KUKA KRL program: EPS_2_25716_MHDR04A_A_20260116015254.src

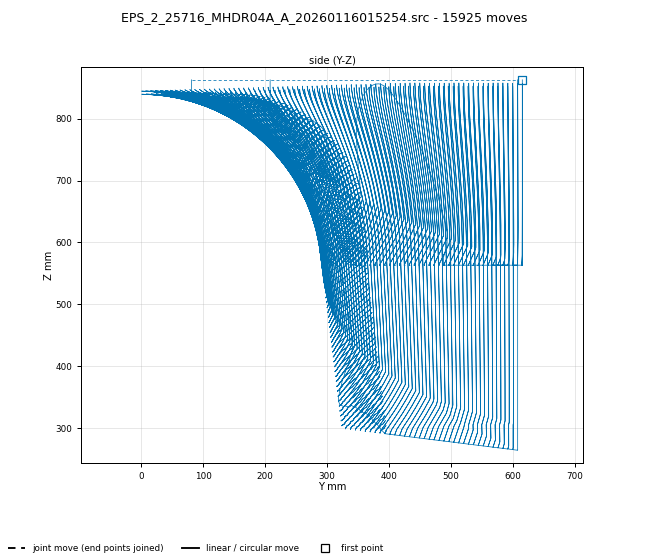
[picture p0: tool path of EPS_2_25716_MHDR04A_A_20260116015254.src, 15925 of 15927 moves have a stored position in this frame; points joined in program order, loops and branches not executed]
&ACCESS RVP
&REL 4
&COMMENT QRS 19112012
&PARAM EDITMASK = *
DEF PART()
EXT BAS (BAS_COMMAND :IN,REAL :IN )
INT I
BAS (#INITMOV,0 )

;KUKA QRS Post kuka4.cps  Date:22-06-2017 !

File_ID=2968

QRS_PRE_INIT()

;Init var - Until changes are made in qrs_pre_init
Outlet_Square_prg=0
Inlet_1_Square_prg=0
Inlet_2_Square_prg=0
Inlet_3_Square_prg=0
Inlet_4_Square_prg=0
Inlet_5_Square_prg=0

Outlet_1={X 0.000, Y 425.000, Z 586.000, B 0.000, E1 0.000 }
Inlet_1={X 0.000, Y 472.270, Z 561.000, B 0.000, E1 180.000 }
Outlet_1_type=533
Inlet_1_type=0
;QRS#1=Sidecore dimensions
;QRS#2=525-21" Concrete
;QRS#3=DeadEnd 533
;QRS#4=
;QRS#5=
;QRS#6=
;QRS#7=
;QRS#8=
;QRS#9=S306-32
;QRS#10=

;QRS#11=
;QRS#12=
;QRS#13=
;QRS#14=
;QRS#15=
;QRS#16=1220x127x1219 4'
;QRS#17=EPS Height
;QRS#18=852,5
;QRS#19=*
;QRS#20= UPDATED VERSION 22-06-2017
;QRS#21=*
Outlet_Square=0250
Inlet_1_Square=00
Inlet_2_Square=0
Inlet_3_Square=0
Inlet_4_Square=0
Inlet_5_Square=0
Mill_Square=1
Outlet_Square_Prg=263
Inlet_1_Square_prg=0

QRS_INIT()

$ADVANCE=5

; T1
PTP {E1 172.624,E2 172.624}
PTP {X 0,Y 615.399,A -85,B 0,C 180,E1 172.624,E2 172.624,E3 0,E4 0,E5 0,E6 0}
QRS_SPEED_INIT()
LIN {X 0,Y 615.399,Z 862.5,A -85,B 0,C 180,E1 172.624,E2 172.624,E3 0,E4 0,E5 0,E6 0} C_VEL
LIN {X 0,Y 615.399,Z 565.28,A -85,B 0,C 180,E1 172.624,E2 172.624} C_VEL
LIN {X 0,Y 615.426,Z 563.28,A -85,B 0,C 180,E1 172.81,E2 172.81} C_VEL
LIN {X 0,Y 615.832,Z 563.28,A -85,B 0,C 180,E1 174.193,E2 174.193} C_VEL
LIN {X 0,Y 615.876,Z 563.28,A -85,B 0,C 180,E1 178.841,E2 178.841} C_VEL
LIN {X 0,Y 615.817,Z 563.28,A -85,B 0,C 180,E1 183.48,E2 183.48} C_VEL
LIN {X 0,Y 615.805,Z 563.28,A -85,B 0,C 180,E1 188.143,E2 188.143} C_VEL
LIN {X 0,Y 615.837,Z 563.28,A -85,B 0,C 180,E1 192.861,E2 192.861} C_VEL
LIN {X 0,Y 615.756,Z 563.28,A -85,B 0,C 180,E1 197.672,E2 197.672} C_VEL
LIN {X 0,Y 615.769,Z 563.28,A -85,B 0,C 180,E1 197.99,E2 197.99} C_VEL
LIN {X 0,Y 615.763,Z 563.28,A -85,B 0,C 180,E1 202.613,E2 202.613} C_VEL
LIN {X 0,Y 615.222,Z 563.28,A -85,B 0,C 180,E1 205.173,E2 205.173} C_VEL
LIN {X 0,Y 615.704,Z 563.28,A -85,B 0,C 180,E1 207.743,E2 207.743} C_VEL
LIN {X 0,Y 615.235,Z 563.28,A -85,B 0,C 180,E1 210.422,E2 210.422} C_VEL
LIN {X 0,Y 615.861,Z 563.28,A -85,B 0,C 180,E1 213.115,E2 213.115} C_VEL
LIN {X 0,Y 615.558,Z 563.28,A -85,B 0,C 180,E1 215.95,E2 215.95} C_VEL
LIN {X 0,Y 615.606,Z 563.28,A -85,B 0,C 180,E1 217.868,E2 217.868} C_VEL
LIN {X 0,Y 615.618,Z 563.28,A -85,B 0,C 180,E1 221.912,E2 221.912} C_VEL
LIN {X 0,Y 615.192,Z 563.28,A -85,B 0,C 180,E1 225.151,E2 225.151} C_VEL
LIN {X 0,Y 615.658,Z 563.28,A -85,B 0,C 180,E1 228.093,E2 228.093} C_VEL
LIN {X 0,Y 615.552,Z 563.28,A -85,B 0,C 180,E1 232.141,E2 232.141} C_VEL
LIN {X 0,Y 615.541,Z 563.28,A -85,B 0,C 180,E1 234.05,E2 234.05} C_VEL
LIN {X 0,Y 615.711,Z 563.28,A -85,B 0,C 180,E1 236.078,E2 236.078} C_VEL
LIN {X 0,Y 615.746,Z 563.28,A -85,B 0,C 180,E1 236.879,E2 236.879} C_VEL
LIN {X 0,Y 615.823,Z 563.28,A -85,B 0,C 180,E1 240.472,E2 240.472} C_VEL
LIN {X 0,Y 615.17,Z 563.28,A -85,B 0,C 180,E1 240.877,E2 240.877} C_VEL
LIN {X 0,Y 614.627,Z 563.28,A -85,B 0,C 180,E1 240.936,E2 240.936} C_VEL
LIN {X 0,Y 614.726,Z 566.395,A -85,B 0,C 180,E1 240.996,E2 240.996} C_VEL
LIN {X 0,Y 615.379,Z 580.016,A -85,B 0,C 180,E1 241.207,E2 241.207} C_VEL
LIN {X 0,Y 615.433,Z 602.784,A -85,B 0,C 180,E1 241.52,E2 241.52} C_VEL
LIN {X 0,Y 615.521,Z 612.728,A -85,B 0,C 180,E1 241.689,E2 241.689} C_VEL
LIN {X 0,Y 615.532,Z 626.222,A -85,B 0,C 180,E1 241.976,E2 241.976} C_VEL
LIN {X 0,Y 615.495,Z 635.643,A -85,B 0,C 180,E1 242.213,E2 242.213} C_VEL
LIN {X 0,Y 615.676,Z 651.537,A -85,B 0,C 180,E1 242.706,E2 242.706} C_VEL
LIN {X 0,Y 615.645,Z 663.962,A -85,B 0,C 180,E1 243.153,E2 243.153} C_VEL
LIN {X 0,Y 615.577,Z 673.88,A -85,B 0,C 180,E1 243.555,E2 243.555} C_VEL
LIN {X 0,Y 615.711,Z 689.6,A -85,B 0,C 180,E1 244.287,E2 244.287} C_VEL
LIN {X 0,Y 615.692,Z 701.948,A -85,B 0,C 180,E1 244.936,E2 244.936} C_VEL
LIN {X 0,Y 615.677,Z 713.617,A -85,B 0,C 180,E1 245.617,E2 245.617} C_VEL
LIN {X 0,Y 615.715,Z 725.413,A -85,B 0,C 180,E1 246.38,E2 246.38} C_VEL
LIN {X 0,Y 615.721,Z 736.092,A -85,B 0,C 180,E1 247.135,E2 247.135} C_VEL
LIN {X 0,Y 615.707,Z 747.395,A -85,B 0,C 180,E1 248.012,E2 248.012} C_VEL
LIN {X 0,Y 615.704,Z 756.656,A -85,B 0,C 180,E1 248.791,E2 248.791} C_VEL
LIN {X 0,Y 615.752,Z 766.793,A -85,B 0,C 180,E1 249.723,E2 249.723} C_VEL
LIN {X 0,Y 615.723,Z 776.057,A -85,B 0,C 180,E1 250.646,E2 250.646} C_VEL
LIN {X 0,Y 615.683,Z 784.416,A -85,B 0,C 180,E1 251.548,E2 251.548} C_VEL
LIN {X 0,Y 615.766,Z 792.777,A -85,B 0,C 180,E1 252.532,E2 252.532} C_VEL
LIN {X 0,Y 615.718,Z 800.682,A -85,B 0,C 180,E1 253.542,E2 253.542} C_VEL
LIN {X 0,Y 615.581,Z 807.427,A -85,B 0,C 180,E1 254.473,E2 254.473} C_VEL
LIN {X 0,Y 615.671,Z 815.061,A -85,B 0,C 180,E1 255.645,E2 255.645} C_VEL
LIN {X 0,Y 615.807,Z 820.438,A -85,B 0,C 180,E1 256.544,E2 256.544} C_VEL
LIN {X 0,Y 615.575,Z 826.91,A -85,B 0,C 180,E1 257.728,E2 257.728} C_VEL
LIN {X 0,Y 615.616,Z 832.624,A -85,B 0,C 180,E1 258.913,E2 258.913} C_VEL
LIN {X 0,Y 615.829,Z 837.634,A -85,B 0,C 180,E1 260.096,E2 260.096} C_VEL
LIN {X 0,Y 615.604,Z 842.064,A -85,B 0,C 180,E1 261.268,E2 261.268} C_VEL
LIN {X 0,Y 615.654,Z 846.465,A -85,B 0,C 180,E1 262.658,E2 262.658} C_VEL
LIN {X 0,Y 615.788,Z 849.368,A -85,B 0,C 180,E1 263.749,E2 263.749} C_VEL
LIN {X 0,Y 615.542,Z 852.381,A -85,B 0,C 180,E1 265.123,E2 265.123} C_VEL
LIN {X 0,Y 615.642,Z 854.591,A -85,B 0,C 180,E1 266.519,E2 266.519} C_VEL
LIN {X 0,Y 615.833,Z 855.667,A -85,B 0,C 180,E1 267.449,E2 267.449} C_VEL
LIN {X 0,Y 615.553,Z 856.715,A -85,B 0,C 180,E1 268.84,E2 268.84} C_VEL
LIN {X 0,Y 615.842,Z 856.659,A -85,B 0,C 180,E1 271.159,E2 271.159} C_VEL
LIN {X 0,Y 615.567,Z 855.717,A -85,B 0,C 180,E1 272.552,E2 272.552} C_VEL
LIN {X 0,Y 615.55,Z 854.608,A -85,B 0,C 180,E1 273.482,E2 273.482} C_VEL
LIN {X 0,Y 615.828,Z 852.329,A -85,B 0,C 180,E1 274.875,E2 274.875} C_VEL
LIN {X 0,Y 615.615,Z 849.405,A -85,B 0,C 180,E1 276.251,E2 276.251} C_VEL
LIN {X 0,Y 615.622,Z 846.265,A -85,B 0,C 180,E1 277.419,E2 277.419} C_VEL
LIN {X 0,Y 615.784,Z 842.036,A -85,B 0,C 180,E1 278.729,E2 278.729} C_VEL
LIN {X 0,Y 615.572,Z 837.671,A -85,B 0,C 180,E1 279.908,E2 279.908} C_VEL
LIN {X 0,Y 615.632,Z 832.622,A -85,B 0,C 180,E1 281.086,E2 281.086} C_VEL
LIN {X 0,Y 615.805,Z 826.883,A -85,B 0,C 180,E1 282.267,E2 282.267} C_VEL
LIN {X 0,Y 615.626,Z 820.456,A -85,B 0,C 180,E1 283.46,E2 283.46} C_VEL
LIN {X 0,Y 615.698,Z 813.195,A -85,B 0,C 180,E1 284.654,E2 284.654} C_VEL
LIN {X 0,Y 615.811,Z 807.631,A -85,B 0,C 180,E1 285.488,E2 285.488} C_VEL
LIN {X 0,Y 615.663,Z 798.199,A -85,B 0,C 180,E1 286.791,E2 286.791} C_VEL
LIN {X 0,Y 615.737,Z 789.606,A -85,B 0,C 180,E1 287.852,E2 287.852} C_VEL
LIN {X 0,Y 615.77,Z 781.414,A -85,B 0,C 180,E1 288.784,E2 288.784} C_VEL
LIN {X 0,Y 615.697,Z 771.526,A -85,B 0,C 180,E1 289.816,E2 289.816} C_VEL
LIN {X 0,Y 615.715,Z 763.539,A -85,B 0,C 180,E1 290.588,E2 290.588} C_VEL
LIN {X 0,Y 615.746,Z 753.036,A -85,B 0,C 180,E1 291.518,E2 291.518} C_VEL
LIN {X 0,Y 615.704,Z 743.049,A -85,B 0,C 180,E1 292.335,E2 292.335} C_VEL
LIN {X 0,Y 615.702,Z 733.298,A -85,B 0,C 180,E1 293.071,E2 293.071} C_VEL
LIN {X 0,Y 615.683,Z 721.635,A -85,B 0,C 180,E1 293.874,E2 293.874} C_VEL
LIN {X 0,Y 615.698,Z 709.596,A -85,B 0,C 180,E1 294.623,E2 294.623} C_VEL
LIN {X 0,Y 615.649,Z 698.891,A -85,B 0,C 180,E1 295.234,E2 295.234} C_VEL
LIN {X 0,Y 615.644,Z 688.027,A -85,B 0,C 180,E1 295.796,E2 295.796} C_VEL
LIN {X 0,Y 615.702,Z 673.88,A -85,B 0,C 180,E1 296.439,E2 296.439} C_VEL
LIN {X 0,Y 615.617,Z 660.684,A -85,B 0,C 180,E1 296.971,E2 296.971} C_VEL
LIN {X 0,Y 615.56,Z 651.537,A -85,B 0,C 180,E1 297.299,E2 297.299} C_VEL
LIN {X 0,Y 615.62,Z 634.846,A -85,B 0,C 180,E1 297.801,E2 297.801} C_VEL
LIN {X 0,Y 615.416,Z 621.524,A -85,B 0,C 180,E1 298.137,E2 298.137} C_VEL
LIN {X 0,Y 615.596,Z 607.658,A -85,B 0,C 180,E1 298.397,E2 298.397} C_VEL
LIN {X 0,Y 615.505,Z 590.993,A -85,B 0,C 180,E1 298.643,E2 298.643} C_VEL
LIN {X 0,Y 615.29,Z 577.557,A -85,B 0,C 180,E1 298.829,E2 298.829} C_VEL
LIN {X 0,Y 614.571,Z 564.121,A -85,B 0,C 180,E1 299.042,E2 299.042} C_VEL
LIN {X 0,Y 614.836,Z 563.28,A -85,B 0,C 180,E1 299.087,E2 299.087} C_VEL
LIN {X 0,Y 615.174,Z 563.28,A -85,B 0,C 180,E1 299.128,E2 299.128} C_VEL
LIN {X 0,Y 615.852,Z 563.28,A -85,B 0,C 180,E1 299.532,E2 299.532} C_VEL
LIN {X 0,Y 615.848,Z 563.28,A -85,B 0,C 180,E1 300.387,E2 300.387} C_VEL
LIN {X 0,Y 615.152,Z 563.28,A -85,B 0,C 180,E1 303.844,E2 303.844} C_VEL
LIN {X 0,Y 615.705,Z 563.28,A -85,B 0,C 180,E1 305.939,E2 305.939} C_VEL
LIN {X 0,Y 615.725,Z 563.28,A -85,B 0,C 180,E1 308.857,E2 308.857} C_VEL
LIN {X 0,Y 615.233,Z 563.28,A -85,B 0,C 180,E1 311.942,E2 311.942} C_VEL
LIN {X 0,Y 615.67,Z 563.28,A -85,B 0,C 180,E1 314.894,E2 314.894} C_VEL
LIN {X 0,Y 615.636,Z 563.28,A -85,B 0,C 180,E1 318.496,E2 318.496} C_VEL
LIN {X 0,Y 615.343,Z 563.28,A -85,B 0,C 180,E1 321.113,E2 321.113} C_VEL
LIN {X 0,Y 615.391,Z 563.28,A -85,B 0,C 180,E1 322.158,E2 322.158} C_VEL
LIN {X 0,Y 615.635,Z 563.28,A -85,B 0,C 180,E1 324.055,E2 324.055} C_VEL
LIN {X 0,Y 615.105,Z 563.28,A -85,B 0,C 180,E1 326.839,E2 326.839} C_VEL
LIN {X 0,Y 615.706,Z 563.28,A -85,B 0,C 180,E1 329.604,E2 329.604} C_VEL
LIN {X 0,Y 615.206,Z 563.28,A -85,B 0,C 180,E1 332.233,E2 332.233} C_VEL
LIN {X 0,Y 615.75,Z 563.28,A -85,B 0,C 180,E1 334.85,E2 334.85} C_VEL
LIN {X 0,Y 615.758,Z 563.28,A -85,B 0,C 180,E1 339.877,E2 339.877} C_VEL
LIN {X 0,Y 615.78,Z 563.28,A -85,B 0,C 180,E1 343.784,E2 343.784} C_VEL
LIN {X 0,Y 615.808,Z 563.28,A -85,B 0,C 180,E1 349.507,E2 349.507} C_VEL
LIN {X 0,Y 615.82,Z 563.28,A -85,B 0,C 180,E1 354.193,E2 354.193} C_VEL
LIN {X 0,Y 615.861,Z 563.28,A -85,B 0,C 180,E1 358.841,E2 358.841} C_VEL
LIN {X 0,Y 615.87,Z 563.28,A -85,B 0,C 180,E1 363.48,E2 363.48} C_VEL
LIN {X 0,Y 615.8,Z 563.28,A -85,B 0,C 180,E1 368.143,E2 368.143} C_VEL
LIN {X 0,Y 615.811,Z 563.28,A -85,B 0,C 180,E1 372.861,E2 372.861} C_VEL
LIN {X 0,Y 615.81,Z 563.28,A -85,B 0,C 180,E1 377.67,E2 377.67} C_VEL
LIN {X 0,Y 615.807,Z 563.28,A -85,B 0,C 180,E1 378.001,E2 378.001} C_VEL
LIN {X 0,Y 615.761,Z 563.28,A -85,B 0,C 180,E1 382.613,E2 382.613} C_VEL
LIN {X 0,Y 615.227,Z 563.28,A -85,B 0,C 180,E1 385.173,E2 385.173} C_VEL
LIN {X 0,Y 615.728,Z 563.28,A -85,B 0,C 180,E1 387.742,E2 387.742} C_VEL
LIN {X 0,Y 615.24,Z 563.28,A -85,B 0,C 180,E1 390.422,E2 390.422} C_VEL
LIN {X 0,Y 615.85,Z 563.28,A -85,B 0,C 180,E1 393.116,E2 393.116} C_VEL
LIN {X 0,Y 615.533,Z 563.28,A -85,B 0,C 180,E1 395.952,E2 395.952} C_VEL
LIN {X 0,Y 615.606,Z 563.28,A -85,B 0,C 180,E1 397.868,E2 397.868} C_VEL
LIN {X 0,Y 615.685,Z 563.28,A -85,B 0,C 180,E1 401.906,E2 401.906} C_VEL
LIN {X 0,Y 615.223,Z 563.28,A -85,B 0,C 180,E1 405.148,E2 405.148} C_VEL
LIN {X 0,Y 615.683,Z 563.28,A -85,B 0,C 180,E1 408.095,E2 408.095} C_VEL
LIN {X 0,Y 615.591,Z 563.28,A -85,B 0,C 180,E1 412.136,E2 412.136} C_VEL
LIN {X 0,Y 615.556,Z 563.28,A -85,B 0,C 180,E1 414.051,E2 414.051} C_VEL
LIN {X 0,Y 615.726,Z 563.28,A -85,B 0,C 180,E1 416.076,E2 416.076} C_VEL
LIN {X 0,Y 615.719,Z 563.28,A -85,B 0,C 180,E1 416.878,E2 416.878} C_VEL
LIN {X 0,Y 615.543,Z 563.28,A -85,B 0,C 180,E1 420.519,E2 420.519} C_VEL
LIN {X 0,Y 615.508,Z 563.28,A -85,B 0,C 180,E1 422.249,E2 422.249} C_VEL
LIN {X 0,Y 615.423,Z 563.28,A -85,B 0,C 180,E1 425.669,E2 425.669} C_VEL
LIN {X 0,Y 615.587,Z 563.28,A -85,B 0,C 180,E1 427.381,E2 427.381} C_VEL
LIN {X 0,Y 615.807,Z 563.28,A -85,B 0,C 180,E1 432.005,E2 432.005} C_VEL
LIN {X 0,Y 615.812,Z 563.28,A -85,B 0,C 180,E1 432.331,E2 432.331} C_VEL
LIN {X 0,Y 615.818,Z 563.28,A -85,B 0,C 180,E1 437.139,E2 437.139} C_VEL
LIN {X 0,Y 615.845,Z 563.28,A -85,B 0,C 180,E1 441.857,E2 441.857} C_VEL
LIN {X 0,Y 615.853,Z 563.28,A -85,B 0,C 180,E1 446.52,E2 446.52} C_VEL
LIN {X 0,Y 615.874,Z 563.28,A -85,B 0,C 180,E1 451.159,E2 451.159} C_VEL
LIN {X 0,Y 615.861,Z 563.28,A -85,B 0,C 180,E1 455.806,E2 455.806} C_VEL
LIN {X 0,Y 615.821,Z 563.28,A -85,B 0,C 180,E1 460.493,E2 460.493} C_VEL
LIN {X 0,Y 615.809,Z 563.28,A -85,B 0,C 180,E1 465.251,E2 465.251} C_VEL
LIN {X 0,Y 615.79,Z 563.28,A -85,B 0,C 180,E1 470.121,E2 470.121} C_VEL
LIN {X 0,Y 615.764,Z 563.28,A -85,B 0,C 180,E1 475.149,E2 475.149} C_VEL
LIN {X 0,Y 615.395,Z 563.28,A -85,B 0,C 180,E1 479.457,E2 479.457} C_VEL
LIN {X 0,Y 615.72,Z 563.28,A -85,B 0,C 180,E1 480.394,E2 480.394} C_VEL
LIN {X 0,Y 615.148,Z 563.28,A -85,B 0,C 180,E1 483.844,E2 483.844} C_VEL
LIN {X 0,Y 615.695,Z 563.28,A -85,B 0,C 180,E1 485.939,E2 485.939} C_VEL
LIN {X 0,Y 615.655,Z 563.28,A -85,B 0,C 180,E1 487.871,E2 487.871} C_VEL
LIN {X 0,Y 615.739,Z 563.28,A -85,B 0,C 180,E1 488.856,E2 488.856} C_VEL
LIN {X 0,Y 615.245,Z 563.28,A -85,B 0,C 180,E1 491.941,E2 491.941} C_VEL
LIN {X 0,Y 615.675,Z 563.28,A -85,B 0,C 180,E1 494.895,E2 494.895} C_VEL
LIN {X 0,Y 615.643,Z 563.28,A -85,B 0,C 180,E1 498.495,E2 498.495} C_VEL
LIN {X 0,Y 615.366,Z 563.28,A -85,B 0,C 180,E1 501.115,E2 501.115} C_VEL
LIN {X 0,Y 615.411,Z 563.28,A -85,B 0,C 180,E1 502.155,E2 502.155} C_VEL
LIN {X 0,Y 615.682,Z 563.28,A -85,B 0,C 180,E1 504.059,E2 504.059} C_VEL
LIN {X 0,Y 615.129,Z 563.28,A -85,B 0,C 180,E1 506.841,E2 506.841} C_VEL
LIN {X 0,Y 615.712,Z 563.28,A -85,B 0,C 180,E1 509.604,E2 509.604} C_VEL
LIN {X 0,Y 615.229,Z 563.28,A -85,B 0,C 180,E1 512.234,E2 512.234} C_VEL
LIN {X 0,Y 615.78,Z 563.28,A -85,B 0,C 180,E1 514.851,E2 514.851} C_VEL
LIN {X 0,Y 615.783,Z 563.28,A -85,B 0,C 180,E1 519.878,E2 519.878} C_VEL
LIN {X 0,Y 615.72,Z 563.28,A -85,B 0,C 180,E1 523.298,E2 523.298} C_VEL
LIN {X 0,Y 615.386,Z 563.28,A -85,B 0,C 180,E1 524.737,E2 524.737} C_VEL
LIN {X 0,Y 615.804,Z 563.28,A -85,B 0,C 180,E1 529.507,E2 529.507} C_VEL
LIN {X 0,Y 615.426,Z 563.28,A -85,B 0,C 180,E1 532.81,E2 532.81} C_VEL
LIN {X 0,Y 613.004,Z 563.28,A -85,B 0,C 180,E1 534.012,E2 534.012} C_VEL
LIN {X 0,Y 607.591,Z 563.28,A -85,B 0,C 180,E1 535.809,E2 535.809} C_VEL
LIN {X 0,Y 607.482,Z 563.28,A -85,B 0,C 180,E1 536.017,E2 536.017} C_VEL
LIN {X 0,Y 607.61,Z 563.28,A -85,B 0,C 180,E1 539.999,E2 539.999} C_VEL
LIN {X 0,Y 607.656,Z 563.28,A -85,B 0,C 180,E1 544.271,E2 544.271} C_VEL
LIN {X 0,Y 607.76,Z 563.28,A -85,B 0,C 180,E1 548.566,E2 548.566} C_VEL
LIN {X 0,Y 607.927,Z 563.28,A -85,B 0,C 180,E1 552.907,E2 552.907} C_VEL
LIN {X 0,Y 607.596,Z 563.28,A -85,B 0,C 180,E1 558.834,E2 558.834} C_VEL
LIN {X 0,Y 607.579,Z 563.28,A -85,B 0,C 180,E1 563.413,E2 563.413} C_VEL
LIN {X 0,Y 607.666,Z 563.28,A -85,B 0,C 180,E1 568.151,E2 568.151} C_VEL
LIN {X 0,Y 607.954,Z 563.28,A -85,B 0,C 180,E1 573.095,E2 573.095} C_VEL
LIN {X 0,Y 607.552,Z 563.28,A -85,B 0,C 180,E1 578.382,E2 578.382} C_VEL
LIN {X 0,Y 607.644,Z 563.28,A -85,B 0,C 180,E1 582.104,E2 582.104} C_VEL
LIN {X 0,Y 607.732,Z 563.28,A -85,B 0,C 180,E1 588.148,E2 588.148} C_VEL
LIN {X 0,Y 607.577,Z 563.28,A -85,B 0,C 180,E1 593.41,E2 593.41} C_VEL
LIN {X 0,Y 607.682,Z 563.28,A -85,B 0,C 180,E1 597.592,E2 597.592} C_VEL
LIN {X 0,Y 607.69,Z 563.28,A -85,B 0,C 180,E1 600.567,E2 600.567} C_VEL
LIN {X 0,Y 608.559,Z 624.797,A -85,B 0,C 180,E1 601.589,E2 601.589} C_VEL
LIN {X 0,Y 608.498,Z 665.533,A -85,B 0,C 180,E1 602.876,E2 602.876} C_VEL
LIN {X 0,Y 608.385,Z 702.866,A -85,B 0,C 180,E1 604.667,E2 604.667} C_VEL
LIN {X 0,Y 608.235,Z 738.17,A -85,B 0,C 180,E1 606.998,E2 606.998} C_VEL
LIN {X 0,Y 608.103,Z 768.949,A -85,B 0,C 180,E1 609.67,E2 609.67} C_VEL
LIN {X 0,Y 608.003,Z 795.695,A -85,B 0,C 180,E1 612.672,E2 612.672} C_VEL
LIN {X 0,Y 607.895,Z 818.344,A -85,B 0,C 180,E1 615.993,E2 615.993} C_VEL
LIN {X 0,Y 607.88,Z 836.513,A -85,B 0,C 180,E1 619.631,E2 619.631} C_VEL
LIN {X 0,Y 607.848,Z 848.574,A -85,B 0,C 180,E1 623.205,E2 623.205} C_VEL
LIN {X 0,Y 607.671,Z 853.956,A -85,B 0,C 180,E1 625.727,E2 625.727} C_VEL
LIN {X 0,Y 607.708,Z 857.086,A -85,B 0,C 180,E1 628.576,E2 628.576} C_VEL
LIN {X 0,Y 607.886,Z 857.087,A -85,B 0,C 180,E1 631.422,E2 631.422} C_VEL
LIN {X 0,Y 607.927,Z 852.758,A -85,B 0,C 180,E1 634.983,E2 634.983} C_VEL
LIN {X 0,Y 607.878,Z 842.075,A -85,B 0,C 180,E1 638.925,E2 638.925} C_VEL
LIN {X 0,Y 607.906,Z 826.455,A -85,B 0,C 180,E1 642.544,E2 642.544} C_VEL
LIN {X 0,Y 607.957,Z 805.351,A -85,B 0,C 180,E1 646.029,E2 646.029} C_VEL
LIN {X 0,Y 608.034,Z 779.03,A -85,B 0,C 180,E1 649.289,E2 649.289} C_VEL
LIN {X 0,Y 608.171,Z 749.03,A -85,B 0,C 180,E1 652.137,E2 652.137} C_VEL
LIN {X 0,Y 608.315,Z 715.907,A -85,B 0,C 180,E1 654.551,E2 654.551} C_VEL
LIN {X 0,Y 608.48,Z 679.749,A -85,B 0,C 180,E1 656.512,E2 656.512} C_VEL
LIN {X 0,Y 608.582,Z 643.016,A -85,B 0,C 180,E1 657.91,E2 657.91} C_VEL
LIN {X 0,Y 608.637,Z 607.158,A -85,B 0,C 180,E1 658.759,E2 658.759} C_VEL
LIN {X 0,Y 607.764,Z 563.28,A -85,B 0,C 180,E1 659.466,E2 659.466} C_VEL
LIN {X 0,Y 607.703,Z 563.28,A -85,B 0,C 180,E1 666.58,E2 666.58} C_VEL
LIN {X 0,Y 607.312,Z 563.28,A -85,B 0,C 180,E1 672.134,E2 672.134} C_VEL
LIN {X 0,Y 607.571,Z 563.28,A -85,B 0,C 180,E1 677.89,E2 677.89} C_VEL
LIN {X 0,Y 607.598,Z 563.28,A -85,B 0,C 180,E1 683.415,E2 683.415} C_VEL
LIN {X 0,Y 607.539,Z 563.28,A -85,B 0,C 180,E1 690.38,E2 690.38} C_VEL
LIN {X 0,Y 607.785,Z 563.28,A -85,B 0,C 180,E1 695.036,E2 695.036} C_VEL
LIN {X 0,Y 607.555,Z 563.28,A -85,B 0,C 180,E1 701.164,E2 701.164} C_VEL
LIN {X 0,Y 607.221,Z 563.28,A -85,B 0,C 180,E1 705.612,E2 705.612} C_VEL
LIN {X 0,Y 607.733,Z 563.28,A -85,B 0,C 180,E1 709.992,E2 709.992} C_VEL
LIN {X 0,Y 607.882,Z 563.28,A -85,B 0,C 180,E1 714.303,E2 714.303} C_VEL
LIN {X 0,Y 607.584,Z 563.28,A -85,B 0,C 180,E1 720.001,E2 720.001} C_VEL
LIN {X 0,Y 607.669,Z 563.28,A -85,B 0,C 180,E1 724.274,E2 724.274} C_VEL
LIN {X 0,Y 607.757,Z 563.28,A -85,B 0,C 180,E1 728.569,E2 728.569} C_VEL
LIN {X 0,Y 607.883,Z 563.28,A -85,B 0,C 180,E1 732.911,E2 732.911} C_VEL
LIN {X 0,Y 607.601,Z 563.28,A -85,B 0,C 180,E1 738.837,E2 738.837} C_VEL
LIN {X 0,Y 607.579,Z 563.28,A -85,B 0,C 180,E1 743.416,E2 743.416} C_VEL
LIN {X 0,Y 607.674,Z 563.28,A -85,B 0,C 180,E1 748.154,E2 748.154} C_VEL
LIN {X 0,Y 607.942,Z 563.28,A -85,B 0,C 180,E1 753.099,E2 753.099} C_VEL
LIN {X 0,Y 607.564,Z 563.28,A -85,B 0,C 180,E1 758.385,E2 758.385} C_VEL
LIN {X 0,Y 607.717,Z 563.28,A -85,B 0,C 180,E1 762.102,E2 762.102} C_VEL
LIN {X 0,Y 607.766,Z 563.28,A -85,B 0,C 180,E1 768.149,E2 768.149} C_VEL
LIN {X 0,Y 607.616,Z 563.28,A -85,B 0,C 180,E1 773.414,E2 773.414} C_VEL
LIN {X 0,Y 607.597,Z 563.28,A -85,B 0,C 180,E1 777.61,E2 777.61} C_VEL
LIN {X 0,Y 607.587,Z 563.28,A -85,B 0,C 180,E1 781.844,E2 781.844} C_VEL
LIN {X 0,Y 607.461,Z 563.28,A -85,B 0,C 180,E1 788.123,E2 788.123} C_VEL
LIN {X 0,Y 607.79,Z 563.28,A -85,B 0,C 180,E1 792.667,E2 792.667} C_VEL
LIN {X 0,Y 607.89,Z 563.28,A -85,B 0,C 180,E1 797.091,E2 797.091} C_VEL
LIN {X 0,Y 607.6,Z 563.28,A -85,B 0,C 180,E1 802.867,E2 802.867} C_VEL
LIN {X 0,Y 607.729,Z 563.28,A -85,B 0,C 180,E1 807.154,E2 807.154} C_VEL
LIN {X 0,Y 607.865,Z 563.28,A -85,B 0,C 180,E1 811.423,E2 811.423} C_VEL
LIN {X 0,Y 607.66,Z 563.28,A -85,B 0,C 180,E1 816.619,E2 816.619} C_VEL
LIN {X 0,Y 607.592,Z 563.28,A -85,B 0,C 180,E1 821.461,E2 821.461} C_VEL
LIN {X 0,Y 607.662,Z 563.28,A -85,B 0,C 180,E1 825.853,E2 825.853} C_VEL
LIN {X 0,Y 607.792,Z 563.28,A -85,B 0,C 180,E1 830.341,E2 830.341} C_VEL
LIN {X 0,Y 607.801,Z 563.28,A -85,B 0,C 180,E1 834.966,E2 834.966} C_VEL
LIN {X 0,Y 607.608,Z 563.28,A -85,B 0,C 180,E1 839.783,E2 839.783} C_VEL
LIN {X 0,Y 607.725,Z 563.28,A -85,B 0,C 180,E1 846.58,E2 846.58} C_VEL
LIN {X 0,Y 607.33,Z 563.28,A -85,B 0,C 180,E1 851.805,E2 851.805} C_VEL
LIN {X 0,Y 607.496,Z 563.28,A -85,B 0,C 180,E1 856.085,E2 856.085} C_VEL
LIN {X 0,Y 607.415,Z 563.28,A -85,B 0,C 180,E1 860.367,E2 860.367} C_VEL
LIN {X 0,Y 607.409,Z 563.28,A -85,B 0,C 180,E1 865.151,E2 865.151} C_VEL
LIN {X 0,Y 607.556,Z 563.28,A -85,B 0,C 180,E1 870.38,E2 870.38} C_VEL
LIN {X 0,Y 607.802,Z 563.28,A -85,B 0,C 180,E1 875.034,E2 875.034} C_VEL
LIN {X 0,Y 607.616,Z 563.28,A -85,B 0,C 180,E1 881.163,E2 881.163} C_VEL
LIN {X 0,Y 607.226,Z 563.28,A -85,B 0,C 180,E1 885.742,E2 885.742} C_VEL
LIN {X 0,Y 607.733,Z 563.28,A -85,B 0,C 180,E1 889.989,E2 889.989} C_VEL
LIN {X 0,Y 607.888,Z 563.28,A -85,B 0,C 180,E1 894.3,E2 894.3} C_VEL
LIN {X 0,Y 607.482,Z 563.28,A -85,B 0,C 180,E1 896.017,E2 896.017} C_VEL
LIN {X 0,Y 603.689,Z 563.28,A -85,B 0,C 180,E1 897.629,E2 897.629} C_VEL
LIN {X 0,Y 599.797,Z 563.28,A -85,B 0,C 180,E1 899.261,E2 899.261} C_VEL
LIN {X 0,Y 599.738,Z 563.28,A -85,B 0,C 180,E1 904.327,E2 904.327} C_VEL
LIN {X 0,Y 599.818,Z 563.28,A -85,B 0,C 180,E1 908.68,E2 908.68} C_VEL
LIN {X 0,Y 599.947,Z 563.28,A -85,B 0,C 180,E1 913.082,E2 913.082} C_VEL
LIN {X 0,Y 599.642,Z 563.28,A -85,B 0,C 180,E1 919.094,E2 919.094} C_VEL
LIN {X 0,Y 599.586,Z 563.28,A -85,B 0,C 180,E1 923.744,E2 923.744} C_VEL
LIN {X 0,Y 599.666,Z 563.28,A -85,B 0,C 180,E1 928.56,E2 928.56} C_VEL
LIN {X 0,Y 599.835,Z 563.28,A -85,B 0,C 180,E1 933.881,E2 933.881} C_VEL
LIN {X 0,Y 599.527,Z 563.28,A -85,B 0,C 180,E1 938.992,E2 938.992} C_VEL
LIN {X 0,Y 599.438,Z 563.28,A -85,B 0,C 180,E1 943.109,E2 943.109} C_VEL
LIN {X 0,Y 599.557,Z 563.28,A -85,B 0,C 180,E1 949.126,E2 949.126} C_VEL
LIN {X 0,Y 599.682,Z 563.28,A -85,B 0,C 180,E1 954.636,E2 954.636} C_VEL
LIN {X 0,Y 599.928,Z 563.28,A -85,B 0,C 180,E1 960.161,E2 960.161} C_VEL
LIN {X 0,Y 601.599,Z 583.884,A -85,B 0,C 180,E1 960.536,E2 960.536} C_VEL
LIN {X 0,Y 601.567,Z 627.343,A -85,B 0,C 180,E1 961.294,E2 961.294} C_VEL
LIN {X 0,Y 601.381,Z 666.029,A -85,B 0,C 180,E1 962.549,E2 962.549} C_VEL
LIN {X 0,Y 601.087,Z 702.885,A -85,B 0,C 180,E1 964.338,E2 964.338} C_VEL
LIN {X 0,Y 600.762,Z 737.804,A -85,B 0,C 180,E1 966.666,E2 966.666} C_VEL
LIN {X 0,Y 600.476,Z 768.952,A -85,B 0,C 180,E1 969.4,E2 969.4} C_VEL
LIN {X 0,Y 600.274,Z 795.697,A -85,B 0,C 180,E1 972.442,E2 972.442} C_VEL
LIN {X 0,Y 600.064,Z 818.354,A -85,B 0,C 180,E1 975.808,E2 975.808} C_VEL
LIN {X 0,Y 599.962,Z 835.869,A -85,B 0,C 180,E1 979.338,E2 979.338} C_VEL
LIN {X 0,Y 599.89,Z 847.677,A -85,B 0,C 180,E1 982.774,E2 982.774} C_VEL
LIN {X 0,Y 599.784,Z 853.958,A -85,B 0,C 180,E1 985.671,E2 985.671} C_VEL
LIN {X 0,Y 599.809,Z 857.088,A -85,B 0,C 180,E1 988.558,E2 988.558} C_VEL
LIN {X 0,Y 599.979,Z 857.088,A -85,B 0,C 180,E1 991.441,E2 991.441} C_VEL
LIN {X 0,Y 600.013,Z 852.757,A -85,B 0,C 180,E1 995.049,E2 995.049} C_VEL
LIN {X 0,Y 599.977,Z 842.076,A -85,B 0,C 180,E1 999.043,E2 999.043} C_VEL
LIN {X 0,Y 600.04,Z 826.459,A -85,B 0,C 180,E1 1002.711,E2 1002.711} C_VEL
LIN {X 0,Y 600.116,Z 804.713,A -85,B 0,C 180,E1 1006.334,E2 1006.334} C_VEL
LIN {X 0,Y 600.366,Z 779.034,A -85,B 0,C 180,E1 1009.545,E2 1009.545} C_VEL
LIN {X 0,Y 600.648,Z 748.454,A -85,B 0,C 180,E1 1012.479,E2 1012.479} C_VEL
LIN {X 0,Y 601.003,Z 713.913,A -85,B 0,C 180,E1 1015,E2 1015} C_VEL
LIN {X 0,Y 601.367,Z 675.827,A -85,B 0,C 180,E1 1017.037,E2 1017.037} C_VEL
LIN {X 0,Y 601.573,Z 636.508,A -85,B 0,C 180,E1 1018.463,E2 1018.463} C_VEL
LIN {X 0,Y 601.717,Z 596.802,A -85,B 0,C 180,E1 1019.285,E2 1019.285} C_VEL
LIN {X 0,Y 600.038,Z 563.28,A -85,B 0,C 180,E1 1019.835,E2 1019.835} C_VEL
LIN {X 0,Y 599.744,Z 563.28,A -85,B 0,C 180,E1 1027.146,E2 1027.146} C_VEL
LIN {X 0,Y 599.412,Z 563.28,A -85,B 0,C 180,E1 1033.111,E2 1033.111} C_VEL
LIN {X 0,Y 599.576,Z 563.28,A -85,B 0,C 180,E1 1039.028,E2 1039.028} C_VEL
LIN {X 0,Y 599.521,Z 563.28,A -85,B 0,C 180,E1 1044.628,E2 1044.628} C_VEL
LIN {X 0,Y 599.594,Z 563.28,A -85,B 0,C 180,E1 1049.781,E2 1049.781} C_VEL
LIN {X 0,Y 599.852,Z 563.28,A -85,B 0,C 180,E1 1054.907,E2 1054.907} C_VEL
LIN {X 0,Y 599.708,Z 563.28,A -85,B 0,C 180,E1 1060.908,E2 1060.908} C_VEL
LIN {X 0,Y 599.36,Z 563.28,A -85,B 0,C 180,E1 1065.42,E2 1065.42} C_VEL
LIN {X 0,Y 599.793,Z 563.28,A -85,B 0,C 180,E1 1069.858,E2 1069.858} C_VEL
LIN {X 0,Y 599.981,Z 563.28,A -85,B 0,C 180,E1 1074.228,E2 1074.228} C_VEL
LIN {X 0,Y 599.684,Z 563.28,A -85,B 0,C 180,E1 1080.002,E2 1080.002} C_VEL
LIN {X 0,Y 599.751,Z 563.28,A -85,B 0,C 180,E1 1084.33,E2 1084.33} C_VEL
LIN {X 0,Y 599.811,Z 563.28,A -85,B 0,C 180,E1 1088.683,E2 1088.683} C_VEL
LIN {X 0,Y 599.909,Z 563.28,A -85,B 0,C 180,E1 1093.086,E2 1093.086} C_VEL
LIN {X 0,Y 599.661,Z 563.28,A -85,B 0,C 180,E1 1099.096,E2 1099.096} C_VEL
LIN {X 0,Y 599.587,Z 563.28,A -85,B 0,C 180,E1 1103.747,E2 1103.747} C_VEL
LIN {X 0,Y 599.675,Z 563.28,A -85,B 0,C 180,E1 1108.563,E2 1108.563} C_VEL
LIN {X 0,Y 599.823,Z 563.28,A -85,B 0,C 180,E1 1113.882,E2 1113.882} C_VEL
LIN {X 0,Y 599.534,Z 563.28,A -85,B 0,C 180,E1 1118.995,E2 1118.995} C_VEL
LIN {X 0,Y 599.493,Z 563.28,A -85,B 0,C 180,E1 1123.117,E2 1123.117} C_VEL
LIN {X 0,Y 599.571,Z 563.28,A -85,B 0,C 180,E1 1129.129,E2 1129.129} C_VEL
LIN {X 0,Y 599.715,Z 563.28,A -85,B 0,C 180,E1 1134.64,E2 1134.64} C_VEL
LIN {X 0,Y 599.597,Z 563.28,A -85,B 0,C 180,E1 1139.779,E2 1139.779} C_VEL
LIN {X 0,Y 599.484,Z 563.28,A -85,B 0,C 180,E1 1144.985,E2 1144.985} C_VEL
LIN {X 0,Y 599.394,Z 563.28,A -85,B 0,C 180,E1 1149.363,E2 1149.363} C_VEL
LIN {X 0,Y 599.552,Z 563.28,A -85,B 0,C 180,E1 1153.928,E2 1153.928} C_VEL
LIN {X 0,Y 599.636,Z 563.28,A -85,B 0,C 180,E1 1158.386,E2 1158.386} C_VEL
LIN {X 0,Y 599.702,Z 563.28,A -85,B 0,C 180,E1 1162.773,E2 1162.773} C_VEL
LIN {X 0,Y 599.84,Z 563.28,A -85,B 0,C 180,E1 1167.117,E2 1167.117} C_VEL
LIN {X 0,Y 599.955,Z 563.28,A -85,B 0,C 180,E1 1171.442,E2 1171.442} C_VEL
LIN {X 0,Y 600.029,Z 563.28,A -85,B 0,C 180,E1 1175.774,E2 1175.774} C_VEL
LIN {X 0,Y 599.651,Z 563.28,A -85,B 0,C 180,E1 1181.615,E2 1181.615} C_VEL
LIN {X 0,Y 599.504,Z 563.28,A -85,B 0,C 180,E1 1186.96,E2 1186.96} C_VEL
LIN {X 0,Y 599.564,Z 563.28,A -85,B 0,C 180,E1 1191.371,E2 1191.371} C_VEL
LIN {X 0,Y 599.788,Z 563.28,A -85,B 0,C 180,E1 1195.323,E2 1195.323} C_VEL
LIN {X 0,Y 599.515,Z 563.28,A -85,B 0,C 180,E1 1201.151,E2 1201.151} C_VEL
LIN {X 0,Y 599.801,Z 563.28,A -85,B 0,C 180,E1 1207.144,E2 1207.144} C_VEL
LIN {X 0,Y 599.44,Z 563.28,A -85,B 0,C 180,E1 1213.109,E2 1213.109} C_VEL
LIN {X 0,Y 599.592,Z 563.28,A -85,B 0,C 180,E1 1219.028,E2 1219.028} C_VEL
LIN {X 0,Y 599.546,Z 563.28,A -85,B 0,C 180,E1 1224.626,E2 1224.626} C_VEL
LIN {X 0,Y 599.609,Z 563.28,A -85,B 0,C 180,E1 1229.778,E2 1229.778} C_VEL
LIN {X 0,Y 599.88,Z 563.28,A -85,B 0,C 180,E1 1234.904,E2 1234.904} C_VEL
LIN {X 0,Y 599.758,Z 563.28,A -85,B 0,C 180,E1 1240.907,E2 1240.907} C_VEL
LIN {X 0,Y 599.367,Z 563.28,A -85,B 0,C 180,E1 1245.417,E2 1245.417} C_VEL
LIN {X 0,Y 599.791,Z 563.28,A -85,B 0,C 180,E1 1249.855,E2 1249.855} C_VEL
LIN {X 0,Y 599.99,Z 563.28,A -85,B 0,C 180,E1 1254.225,E2 1254.225} C_VEL
LIN {X 0,Y 599.797,Z 563.28,A -85,B 0,C 180,E1 1259.261,E2 1259.261} C_VEL
LIN {X 0,Y 595.628,Z 563.28,A -85,B 0,C 180,E1 1260.891,E2 1260.891} C_VEL
LIN {X 0,Y 591.8,Z 563.28,A -85,B 0,C 180,E1 1262.544,E2 1262.544} C_VEL
LIN {X 0,Y 591.879,Z 563.28,A -85,B 0,C 180,E1 1268.797,E2 1268.797} C_VEL
LIN {X 0,Y 591.688,Z 563.28,A -85,B 0,C 180,E1 1274.27,E2 1274.27} C_VEL
LIN {X 0,Y 591.703,Z 563.28,A -85,B 0,C 180,E1 1279.36,E2 1279.36} C_VEL
LIN {X 0,Y 591.615,Z 563.28,A -85,B 0,C 180,E1 1284.084,E2 1284.084} C_VEL
LIN {X 0,Y 591.654,Z 563.28,A -85,B 0,C 180,E1 1288.984,E2 1288.984} C_VEL
LIN {X 0,Y 591.905,Z 563.28,A -85,B 0,C 180,E1 1294.114,E2 1294.114} C_VEL
LIN {X 0,Y 591.569,Z 563.28,A -85,B 0,C 180,E1 1300.069,E2 1300.069} C_VEL
LIN {X 0,Y 591.396,Z 563.28,A -85,B 0,C 180,E1 1305.595,E2 1305.595} C_VEL
LIN {X 0,Y 591.55,Z 563.28,A -85,B 0,C 180,E1 1310.376,E2 1310.376} C_VEL
LIN {X 0,Y 591.878,Z 563.28,A -85,B 0,C 180,E1 1315.881,E2 1315.881} C_VEL
LIN {X 0,Y 591.939,Z 563.28,A -85,B 0,C 180,E1 1319.71,E2 1319.71} C_VEL
LIN {X 0,Y 594.223,Z 571.9,A -85,B 0,C 180,E1 1319.969,E2 1319.969} C_VEL
LIN {X 0,Y 594.64,Z 625.616,A -85,B 0,C 180,E1 1320.882,E2 1320.882} C_VEL
LIN {X 0,Y 594.355,Z 664.669,A -85,B 0,C 180,E1 1322.14,E2 1322.14} C_VEL
LIN {X 0,Y 593.831,Z 702.877,A -85,B 0,C 180,E1 1324.001,E2 1324.001} C_VEL
LIN {X 0,Y 593.296,Z 737.639,A -85,B 0,C 180,E1 1326.341,E2 1326.341} C_VEL
LIN {X 0,Y 592.86,Z 768.955,A -85,B 0,C 180,E1 1329.123,E2 1329.123} C_VEL
LIN {X 0,Y 592.532,Z 795.699,A -85,B 0,C 180,E1 1332.205,E2 1332.205} C_VEL
LIN {X 0,Y 592.202,Z 817.821,A -85,B 0,C 180,E1 1335.523,E2 1335.523} C_VEL
LIN {X 0,Y 592.024,Z 834.249,A -85,B 0,C 180,E1 1338.801,E2 1338.801} C_VEL
LIN {X 0,Y 591.971,Z 846.717,A -85,B 0,C 180,E1 1342.308,E2 1342.308} C_VEL
LIN {X 0,Y 591.883,Z 853.961,A -85,B 0,C 180,E1 1345.613,E2 1345.613} C_VEL
LIN {X 0,Y 591.91,Z 857.089,A -85,B 0,C 180,E1 1348.538,E2 1348.538} C_VEL
LIN {X 0,Y 592.073,Z 857.09,A -85,B 0,C 180,E1 1351.46,E2 1351.46} C_VEL
LIN {X 0,Y 592.111,Z 852.754,A -85,B 0,C 180,E1 1355.117,E2 1355.117} C_VEL
LIN {X 0,Y 592.092,Z 842.077,A -85,B 0,C 180,E1 1359.165,E2 1359.165} C_VEL
LIN {X 0,Y 592.188,Z 826.463,A -85,B 0,C 180,E1 1362.883,E2 1362.883} C_VEL
LIN {X 0,Y 592.351,Z 804.942,A -85,B 0,C 180,E1 1366.521,E2 1366.521} C_VEL
LIN {X 0,Y 592.684,Z 778.952,A -85,B 0,C 180,E1 1369.818,E2 1369.818} C_VEL
LIN {X 0,Y 593.107,Z 748.756,A -85,B 0,C 180,E1 1372.754,E2 1372.754} C_VEL
LIN {X 0,Y 593.673,Z 714.69,A -85,B 0,C 180,E1 1375.28,E2 1375.28} C_VEL
LIN {X 0,Y 594.193,Z 676.866,A -85,B 0,C 180,E1 1377.34,E2 1377.34} C_VEL
LIN {X 0,Y 594.596,Z 637.688,A -85,B 0,C 180,E1 1378.793,E2 1378.793} C_VEL
LIN {X 0,Y 594.833,Z 598.877,A -85,B 0,C 180,E1 1379.626,E2 1379.626} C_VEL
LIN {X 0,Y 593.644,Z 568.062,A -85,B 0,C 180,E1 1380.116,E2 1380.116} C_VEL
LIN {X 0,Y 591.957,Z 563.28,A -85,B 0,C 180,E1 1380.332,E2 1380.332} C_VEL
LIN {X 0,Y 591.754,Z 563.28,A -85,B 0,C 180,E1 1385.909,E2 1385.909} C_VEL
LIN {X 0,Y 591.455,Z 563.28,A -85,B 0,C 180,E1 1391.555,E2 1391.555} C_VEL
LIN {X 0,Y 591.616,Z 563.28,A -85,B 0,C 180,E1 1396.477,E2 1396.477} C_VEL
LIN {X 0,Y 591.655,Z 563.28,A -85,B 0,C 180,E1 1402.26,E2 1402.26} C_VEL
LIN {X 0,Y 591.423,Z 563.28,A -85,B 0,C 180,E1 1407.603,E2 1407.603} C_VEL
LIN {X 0,Y 591.535,Z 563.28,A -85,B 0,C 180,E1 1412.668,E2 1412.668} C_VEL
LIN {X 0,Y 591.496,Z 563.28,A -85,B 0,C 180,E1 1417.502,E2 1417.502} C_VEL
LIN {X 0,Y 591.757,Z 563.28,A -85,B 0,C 180,E1 1422.183,E2 1422.183} C_VEL
LIN {X 0,Y 591.597,Z 563.28,A -85,B 0,C 180,E1 1428.227,E2 1428.227} C_VEL
LIN {X 0,Y 592.046,Z 563.28,A -85,B 0,C 180,E1 1434.15,E2 1434.15} C_VEL
LIN {X 0,Y 591.783,Z 563.28,A -85,B 0,C 180,E1 1440.002,E2 1440.002} C_VEL
LIN {X 0,Y 591.834,Z 563.28,A -85,B 0,C 180,E1 1444.388,E2 1444.388} C_VEL
LIN {X 0,Y 591.869,Z 563.28,A -85,B 0,C 180,E1 1448.801,E2 1448.801} C_VEL
LIN {X 0,Y 591.677,Z 563.28,A -85,B 0,C 180,E1 1454.272,E2 1454.272} C_VEL
LIN {X 0,Y 591.706,Z 563.28,A -85,B 0,C 180,E1 1459.363,E2 1459.363} C_VEL
LIN {X 0,Y 591.622,Z 563.28,A -85,B 0,C 180,E1 1464.087,E2 1464.087} C_VEL
LIN {X 0,Y 591.663,Z 563.28,A -85,B 0,C 180,E1 1468.987,E2 1468.987} C_VEL
LIN {X 0,Y 591.895,Z 563.28,A -85,B 0,C 180,E1 1474.118,E2 1474.118} C_VEL
LIN {X 0,Y 591.591,Z 563.28,A -85,B 0,C 180,E1 1480.074,E2 1480.074} C_VEL
LIN {X 0,Y 591.413,Z 563.28,A -85,B 0,C 180,E1 1485.598,E2 1485.598} C_VEL
LIN {X 0,Y 591.569,Z 563.28,A -85,B 0,C 180,E1 1490.379,E2 1490.379} C_VEL
LIN {X 0,Y 591.878,Z 563.28,A -85,B 0,C 180,E1 1495.883,E2 1495.883} C_VEL
LIN {X 0,Y 591.716,Z 563.28,A -85,B 0,C 180,E1 1501.018,E2 1501.018} C_VEL
LIN {X 0,Y 591.638,Z 563.28,A -85,B 0,C 180,E1 1507.507,E2 1507.507} C_VEL
LIN {X 0,Y 591.875,Z 563.28,A -85,B 0,C 180,E1 1512.186,E2 1512.186} C_VEL
LIN {X 0,Y 591.748,Z 563.28,A -85,B 0,C 180,E1 1518.229,E2 1518.229} C_VEL
LIN {X 0,Y 591.823,Z 563.28,A -85,B 0,C 180,E1 1522.676,E2 1522.676} C_VEL
LIN {X 0,Y 591.932,Z 563.28,A -85,B 0,C 180,E1 1527.078,E2 1527.078} C_VEL
LIN {X 0,Y 592.045,Z 563.28,A -85,B 0,C 180,E1 1531.461,E2 1531.461} C_VEL
LIN {X 0,Y 591.975,Z 563.28,A -85,B 0,C 180,E1 1536.194,E2 1536.194} C_VEL
LIN {X 0,Y 591.716,Z 563.28,A -85,B 0,C 180,E1 1541.773,E2 1541.773} C_VEL
LIN {X 0,Y 591.751,Z 563.28,A -85,B 0,C 180,E1 1546.291,E2 1546.291} C_VEL
LIN {X 0,Y 591.795,Z 563.28,A -85,B 0,C 180,E1 1550.916,E2 1550.916} C_VEL
LIN {X 0,Y 591.531,Z 563.28,A -85,B 0,C 180,E1 1556.764,E2 1556.764} C_VEL
LIN {X 0,Y 591.643,Z 563.28,A -85,B 0,C 180,E1 1560.672,E2 1560.672} C_VEL
LIN {X 0,Y 591.771,Z 563.28,A -85,B 0,C 180,E1 1565.91,E2 1565.91} C_VEL
LIN {X 0,Y 591.597,Z 563.28,A -85,B 0,C 180,E1 1570.072,E2 1570.072} C_VEL
LIN {X 0,Y 591.606,Z 563.28,A -85,B 0,C 180,E1 1575.578,E2 1575.578} C_VEL
LIN {X 0,Y 591.575,Z 563.28,A -85,B 0,C 180,E1 1580.378,E2 1580.378} C_VEL
LIN {X 0,Y 591.457,Z 563.28,A -85,B 0,C 180,E1 1585.853,E2 1585.853} C_VEL
LIN {X 0,Y 591.566,Z 563.28,A -85,B 0,C 180,E1 1591.008,E2 1591.008} C_VEL
LIN {X 0,Y 591.677,Z 563.28,A -85,B 0,C 180,E1 1595.916,E2 1595.916} C_VEL
LIN {X 0,Y 591.854,Z 563.28,A -85,B 0,C 180,E1 1600.642,E2 1600.642} C_VEL
LIN {X 0,Y 591.431,Z 563.28,A -85,B 0,C 180,E1 1605.828,E2 1605.828} C_VEL
LIN {X 0,Y 591.659,Z 563.28,A -85,B 0,C 180,E1 1611.196,E2 1611.196} C_VEL
LIN {X 0,Y 591.73,Z 563.28,A -85,B 0,C 180,E1 1615.611,E2 1615.611} C_VEL
LIN {X 0,Y 591.808,Z 563.28,A -85,B 0,C 180,E1 1619.998,E2 1619.998} C_VEL
LIN {X 0,Y 591.8,Z 563.28,A -85,B 0,C 180,E1 1622.544,E2 1622.544} C_VEL
LIN {X 0,Y 589.356,Z 563.28,A -85,B 0,C 180,E1 1623.794,E2 1623.794} C_VEL
LIN {X 0,Y 583.86,Z 563.28,A -85,B 0,C 180,E1 1625.662,E2 1625.662} C_VEL
LIN {X 0,Y 583.768,Z 563.28,A -85,B 0,C 180,E1 1625.879,E2 1625.879} C_VEL
LIN {X 0,Y 583.753,Z 563.28,A -85,B 0,C 180,E1 1630.791,E2 1630.791} C_VEL
LIN {X 0,Y 583.699,Z 563.28,A -85,B 0,C 180,E1 1634.981,E2 1634.981} C_VEL
LIN {X 0,Y 583.76,Z 563.28,A -85,B 0,C 180,E1 1639.634,E2 1639.634} C_VEL
LIN {X 0,Y 583.655,Z 563.28,A -85,B 0,C 180,E1 1644.434,E2 1644.434} C_VEL
LIN {X 0,Y 583.675,Z 563.28,A -85,B 0,C 180,E1 1649.418,E2 1649.418} C_VEL
LIN {X 0,Y 583.913,Z 563.28,A -85,B 0,C 180,E1 1654.646,E2 1654.646} C_VEL
LIN {X 0,Y 583.65,Z 563.28,A -85,B 0,C 180,E1 1660.265,E2 1660.265} C_VEL
LIN {X 0,Y 583.587,Z 563.28,A -85,B 0,C 180,E1 1666.383,E2 1666.383} C_VEL
LIN {X 0,Y 583.701,Z 563.28,A -85,B 0,C 180,E1 1671.65,E2 1671.65} C_VEL
LIN {X 0,Y 583.943,Z 563.28,A -85,B 0,C 180,E1 1677.133,E2 1677.133} C_VEL
LIN {X 0,Y 583.961,Z 563.452,A -85,B 0,C 180,E1 1679.267,E2 1679.267} C_VEL
LIN {X 0,Y 587.456,Z 574.076,A -85,B 0,C 180,E1 1679.617,E2 1679.617} C_VEL
LIN {X 0,Y 587.687,Z 627.043,A -85,B 0,C 180,E1 1680.542,E2 1680.542} C_VEL
LIN {X 0,Y 587.236,Z 666.362,A -85,B 0,C 180,E1 1681.844,E2 1681.844} C_VEL
LIN {X 0,Y 586.564,Z 703.661,A -85,B 0,C 180,E1 1683.702,E2 1683.702} C_VEL
LIN {X 0,Y 585.845,Z 739.127,A -85,B 0,C 180,E1 1686.141,E2 1686.141} C_VEL
LIN {X 0,Y 585.24,Z 770.868,A -85,B 0,C 180,E1 1689.037,E2 1689.037} C_VEL
LIN {X 0,Y 584.748,Z 799.098,A -85,B 0,C 180,E1 1692.412,E2 1692.412} C_VEL
LIN {X 0,Y 584.413,Z 821.651,A -85,B 0,C 180,E1 1696.008,E2 1696.008} C_VEL
LIN {X 0,Y 584.28,Z 839.395,A -85,B 0,C 180,E1 1699.96,E2 1699.96} C_VEL
LIN {X 0,Y 584.186,Z 850.238,A -85,B 0,C 180,E1 1703.595,E2 1703.595} C_VEL
LIN {X 0,Y 584.179,Z 855.914,A -85,B 0,C 180,E1 1707.038,E2 1707.038} C_VEL
LIN {X 0,Y 584.049,Z 857.5,A -85,B 0,C 180,E1 1709.999,E2 1709.999} C_VEL
LIN {X 0,Y 584.028,Z 855.916,A -85,B 0,C 180,E1 1712.961,E2 1712.961} C_VEL
LIN {X 0,Y 584.084,Z 850.416,A -85,B 0,C 180,E1 1716.321,E2 1716.321} C_VEL
LIN {X 0,Y 584.07,Z 839.4,A -85,B 0,C 180,E1 1720.043,E2 1720.043} C_VEL
LIN {X 0,Y 584.312,Z 823.098,A -85,B 0,C 180,E1 1723.713,E2 1723.713} C_VEL
LIN {X 0,Y 584.617,Z 801.435,A -85,B 0,C 180,E1 1727.254,E2 1727.254} C_VEL
LIN {X 0,Y 585.107,Z 774.63,A -85,B 0,C 180,E1 1730.572,E2 1730.572} C_VEL
LIN {X 0,Y 585.773,Z 742.716,A -85,B 0,C 180,E1 1733.572,E2 1733.572} C_VEL
LIN {X 0,Y 586.434,Z 708.106,A -85,B 0,C 180,E1 1736.033,E2 1736.033} C_VEL
LIN {X 0,Y 587.138,Z 670.855,A -85,B 0,C 180,E1 1737.966,E2 1737.966} C_VEL
LIN {X 0,Y 587.65,Z 632.307,A -85,B 0,C 180,E1 1739.319,E2 1739.319} C_VEL
LIN {X 0,Y 587.896,Z 590.604,A -85,B 0,C 180,E1 1740.129,E2 1740.129} C_VEL
LIN {X 0,Y 586.641,Z 570.661,A -85,B 0,C 180,E1 1740.477,E2 1740.477} C_VEL
LIN {X 0,Y 583.929,Z 563.28,A -85,B 0,C 180,E1 1740.744,E2 1740.744} C_VEL
LIN {X 0,Y 583.826,Z 563.28,A -85,B 0,C 180,E1 1746.754,E2 1746.754} C_VEL
LIN {X 0,Y 583.553,Z 563.28,A -85,B 0,C 180,E1 1752.247,E2 1752.247} C_VEL
LIN {X 0,Y 583.72,Z 563.28,A -85,B 0,C 180,E1 1757.77,E2 1757.77} C_VEL
LIN {X 0,Y 583.708,Z 563.28,A -85,B 0,C 180,E1 1763.519,E2 1763.519} C_VEL
LIN {X 0,Y 583.624,Z 563.28,A -85,B 0,C 180,E1 1768.863,E2 1768.863} C_VEL
LIN {X 0,Y 583.819,Z 563.28,A -85,B 0,C 180,E1 1774.775,E2 1774.775} C_VEL
LIN {X 0,Y 583.9,Z 563.28,A -85,B 0,C 180,E1 1780.371,E2 1780.371} C_VEL
LIN {X 0,Y 583.621,Z 563.28,A -85,B 0,C 180,E1 1785.017,E2 1785.017} C_VEL
LIN {X 0,Y 583.919,Z 563.28,A -85,B 0,C 180,E1 1789.58,E2 1789.58} C_VEL
LIN {X 0,Y 584.129,Z 563.28,A -85,B 0,C 180,E1 1794.07,E2 1794.07} C_VEL
LIN {X 0,Y 583.905,Z 563.28,A -85,B 0,C 180,E1 1800.002,E2 1800.002} C_VEL
LIN {X 0,Y 583.933,Z 563.28,A -85,B 0,C 180,E1 1804.448,E2 1804.448} C_VEL
LIN {X 0,Y 583.932,Z 563.28,A -85,B 0,C 180,E1 1808.921,E2 1808.921} C_VEL
LIN {X 0,Y 583.997,Z 563.28,A -85,B 0,C 180,E1 1813.449,E2 1813.449} C_VEL
LIN {X 0,Y 583.942,Z 563.28,A -85,B 0,C 180,E1 1818.067,E2 1818.067} C_VEL
LIN {X 0,Y 583.821,Z 563.28,A -85,B 0,C 180,E1 1822.813,E2 1822.813} C_VEL
LIN {X 0,Y 583.727,Z 563.28,A -85,B 0,C 180,E1 1828.486,E2 1828.486} C_VEL
LIN {X 0,Y 583.908,Z 563.28,A -85,B 0,C 180,E1 1834.651,E2 1834.651} C_VEL
LIN {X 0,Y 583.676,Z 563.28,A -85,B 0,C 180,E1 1840.267,E2 1840.267} C_VEL
LIN {X 0,Y 583.604,Z 563.28,A -85,B 0,C 180,E1 1846.386,E2 1846.386} C_VEL
LIN {X 0,Y 583.723,Z 563.28,A -85,B 0,C 180,E1 1851.653,E2 1851.653} C_VEL
LIN {X 0,Y 583.877,Z 563.28,A -85,B 0,C 180,E1 1857.131,E2 1857.131} C_VEL
LIN {X 0,Y 583.672,Z 563.28,A -85,B 0,C 180,E1 1862.267,E2 1862.267} C_VEL
LIN {X 0,Y 583.73,Z 563.28,A -85,B 0,C 180,E1 1867.185,E2 1867.185} C_VEL
LIN {X 0,Y 583.815,Z 563.28,A -85,B 0,C 180,E1 1873.482,E2 1873.482} C_VEL
LIN {X 0,Y 583.862,Z 563.28,A -85,B 0,C 180,E1 1878.068,E2 1878.068} C_VEL
LIN {X 0,Y 583.917,Z 563.28,A -85,B 0,C 180,E1 1882.577,E2 1882.577} C_VEL
LIN {X 0,Y 584.048,Z 563.28,A -85,B 0,C 180,E1 1887.039,E2 1887.039} C_VEL
LIN {X 0,Y 584.154,Z 563.28,A -85,B 0,C 180,E1 1891.481,E2 1891.481} C_VEL
LIN {X 0,Y 584.172,Z 563.28,A -85,B 0,C 180,E1 1895.931,E2 1895.931} C_VEL
LIN {X 0,Y 583.803,Z 563.28,A -85,B 0,C 180,E1 1901.935,E2 1901.935} C_VEL
LIN {X 0,Y 583.735,Z 563.28,A -85,B 0,C 180,E1 1906.963,E2 1906.963} C_VEL
LIN {X 0,Y 583.752,Z 563.28,A -85,B 0,C 180,E1 1911.469,E2 1911.469} C_VEL
LIN {X 0,Y 583.772,Z 563.28,A -85,B 0,C 180,E1 1916.069,E2 1916.069} C_VEL
LIN {X 0,Y 583.589,Z 563.28,A -85,B 0,C 180,E1 1921.427,E2 1921.427} C_VEL
LIN {X 0,Y 583.861,Z 563.28,A -85,B 0,C 180,E1 1926.753,E2 1926.753} C_VEL
LIN {X 0,Y 583.571,Z 563.28,A -85,B 0,C 180,E1 1932.247,E2 1932.247} C_VEL
LIN {X 0,Y 583.739,Z 563.28,A -85,B 0,C 180,E1 1937.768,E2 1937.768} C_VEL
LIN {X 0,Y 583.726,Z 563.28,A -85,B 0,C 180,E1 1943.516,E2 1943.516} C_VEL
LIN {X 0,Y 583.641,Z 563.28,A -85,B 0,C 180,E1 1948.861,E2 1948.861} C_VEL
LIN {X 0,Y 583.819,Z 563.28,A -85,B 0,C 180,E1 1954.778,E2 1954.778} C_VEL
LIN {X 0,Y 583.924,Z 563.28,A -85,B 0,C 180,E1 1960.368,E2 1960.368} C_VEL
LIN {X 0,Y 583.613,Z 563.28,A -85,B 0,C 180,E1 1965.014,E2 1965.014} C_VEL
LIN {X 0,Y 583.913,Z 563.28,A -85,B 0,C 180,E1 1969.576,E2 1969.576} C_VEL
LIN {X 0,Y 584.14,Z 563.28,A -85,B 0,C 180,E1 1974.067,E2 1974.067} C_VEL
LIN {X 0,Y 583.929,Z 563.28,A -85,B 0,C 180,E1 1979.998,E2 1979.998} C_VEL
LIN {X 0,Y 583.92,Z 563.28,A -85,B 0,C 180,E1 1984.445,E2 1984.445} C_VEL
LIN {X 0,Y 583.768,Z 563.28,A -85,B 0,C 180,E1 1985.879,E2 1985.879} C_VEL
LIN {X 0,Y 579.98,Z 563.28,A -85,B 0,C 180,E1 1987.557,E2 1987.557} C_VEL
LIN {X 0,Y 575.976,Z 563.28,A -85,B 0,C 180,E1 1989.258,E2 1989.258} C_VEL
LIN {X 0,Y 575.942,Z 563.28,A -85,B 0,C 180,E1 1994.202,E2 1994.202} C_VEL
LIN {X 0,Y 575.845,Z 563.28,A -85,B 0,C 180,E1 1999.915,E2 1999.915} C_VEL
LIN {X 0,Y 575.727,Z 563.28,A -85,B 0,C 180,E1 2004.793,E2 2004.793} C_VEL
LIN {X 0,Y 575.722,Z 563.28,A -85,B 0,C 180,E1 2010.121,E2 2010.121} C_VEL
LIN {X 0,Y 575.91,Z 563.28,A -85,B 0,C 180,E1 2015.199,E2 2015.199} C_VEL
LIN {X 0,Y 575.735,Z 563.28,A -85,B 0,C 180,E1 2020.936,E2 2020.936} C_VEL
LIN {X 0,Y 575.748,Z 563.28,A -85,B 0,C 180,E1 2027.208,E2 2027.208} C_VEL
LIN {X 0,Y 575.85,Z 563.28,A -85,B 0,C 180,E1 2032.935,E2 2032.935} C_VEL
LIN {X 0,Y 576.012,Z 563.28,A -85,B 0,C 180,E1 2038.782,E2 2038.782} C_VEL
LIN {X 0,Y 580.72,Z 576.439,A -85,B 0,C 180,E1 2039.26,E2 2039.26} C_VEL
LIN {X 0,Y 580.802,Z 627.058,A -85,B 0,C 180,E1 2040.157,E2 2040.157} C_VEL
LIN {X 0,Y 580.223,Z 665.514,A -85,B 0,C 180,E1 2041.437,E2 2041.437} C_VEL
LIN {X 0,Y 579.406,Z 702.12,A -85,B 0,C 180,E1 2043.255,E2 2043.255} C_VEL
LIN {X 0,Y 578.475,Z 738.03,A -85,B 0,C 180,E1 2045.728,E2 2045.728} C_VEL
LIN {X 0,Y 577.671,Z 768.961,A -85,B 0,C 180,E1 2048.548,E2 2048.548} C_VEL
LIN {X 0,Y 576.998,Z 797.152,A -85,B 0,C 180,E1 2051.904,E2 2051.904} C_VEL
LIN {X 0,Y 576.592,Z 820.887,A -85,B 0,C 180,E1 2055.672,E2 2055.672} C_VEL
LIN {X 0,Y 576.372,Z 838.034,A -85,B 0,C 180,E1 2059.439,E2 2059.439} C_VEL
LIN {X 0,Y 576.269,Z 849.588,A -85,B 0,C 180,E1 2063.232,E2 2063.232} C_VEL
LIN {X 0,Y 576.267,Z 855.917,A -85,B 0,C 180,E1 2066.997,E2 2066.997} C_VEL
LIN {X 0,Y 576.149,Z 857.5,A -85,B 0,C 180,E1 2069.999,E2 2069.999} C_VEL
LIN {X 0,Y 576.127,Z 855.919,A -85,B 0,C 180,E1 2073.002,E2 2073.002} C_VEL
LIN {X 0,Y 576.185,Z 849.591,A -85,B 0,C 180,E1 2076.768,E2 2076.768} C_VEL
LIN {X 0,Y 576.232,Z 838.039,A -85,B 0,C 180,E1 2080.562,E2 2080.562} C_VEL
LIN {X 0,Y 576.496,Z 821.022,A -85,B 0,C 180,E1 2084.305,E2 2084.305} C_VEL
LIN {X 0,Y 576.922,Z 798.691,A -85,B 0,C 180,E1 2087.891,E2 2087.891} C_VEL
LIN {X 0,Y 577.575,Z 770.886,A -85,B 0,C 180,E1 2091.253,E2 2091.253} C_VEL
LIN {X 0,Y 578.388,Z 739.454,A -85,B 0,C 180,E1 2094.159,E2 2094.159} C_VEL
LIN {X 0,Y 579.259,Z 705.067,A -85,B 0,C 180,E1 2096.569,E2 2096.569} C_VEL
LIN {X 0,Y 580.11,Z 668.457,A -85,B 0,C 180,E1 2098.441,E2 2098.441} C_VEL
LIN {X 0,Y 580.692,Z 628.49,A -85,B 0,C 180,E1 2099.81,E2 2099.81} C_VEL
LIN {X 0,Y 580.882,Z 580.011,A -85,B 0,C 180,E1 2100.68,E2 2100.68} C_VEL
LIN {X 0,Y 579.545,Z 572.314,A -85,B 0,C 180,E1 2100.867,E2 2100.867} C_VEL
LIN {X 0,Y 575.891,Z 563.28,A -85,B 0,C 180,E1 2101.257,E2 2101.257} C_VEL
LIN {X 0,Y 575.913,Z 563.28,A -85,B 0,C 180,E1 2107.059,E2 2107.059} C_VEL
LIN {X 0,Y 575.66,Z 563.28,A -85,B 0,C 180,E1 2112.964,E2 2112.964} C_VEL
LIN {X 0,Y 575.787,Z 563.28,A -85,B 0,C 180,E1 2119.069,E2 2119.069} C_VEL
LIN {X 0,Y 575.664,Z 563.28,A -85,B 0,C 180,E1 2124.784,E2 2124.784} C_VEL
LIN {X 0,Y 575.709,Z 563.28,A -85,B 0,C 180,E1 2130.134,E2 2130.134} C_VEL
LIN {X 0,Y 575.866,Z 563.28,A -85,B 0,C 180,E1 2135.214,E2 2135.214} C_VEL
LIN {X 0,Y 575.984,Z 563.28,A -85,B 0,C 180,E1 2140.587,E2 2140.587} C_VEL
LIN {X 0,Y 575.763,Z 563.28,A -85,B 0,C 180,E1 2144.808,E2 2144.808} C_VEL
LIN {X 0,Y 575.876,Z 563.28,A -85,B 0,C 180,E1 2150.956,E2 2150.956} C_VEL
LIN {X 0,Y 575.941,Z 563.28,A -85,B 0,C 180,E1 2155.493,E2 2155.493} C_VEL
LIN {X 0,Y 576.004,Z 563.28,A -85,B 0,C 180,E1 2160.002,E2 2160.002} C_VEL
LIN {X 0,Y 576.018,Z 563.28,A -85,B 0,C 180,E1 2164.509,E2 2164.509} C_VEL
LIN {X 0,Y 576.012,Z 563.28,A -85,B 0,C 180,E1 2169.045,E2 2169.045} C_VEL
LIN {X 0,Y 575.927,Z 563.28,A -85,B 0,C 180,E1 2174.202,E2 2174.202} C_VEL
LIN {X 0,Y 575.852,Z 563.28,A -85,B 0,C 180,E1 2179.919,E2 2179.919} C_VEL
LIN {X 0,Y 575.734,Z 563.28,A -85,B 0,C 180,E1 2184.796,E2 2184.796} C_VEL
LIN {X 0,Y 575.729,Z 563.28,A -85,B 0,C 180,E1 2190.125,E2 2190.125} C_VEL
LIN {X 0,Y 575.907,Z 563.28,A -85,B 0,C 180,E1 2195.203,E2 2195.203} C_VEL
LIN {X 0,Y 575.802,Z 563.28,A -85,B 0,C 180,E1 2200.934,E2 2200.934} C_VEL
LIN {X 0,Y 575.766,Z 563.28,A -85,B 0,C 180,E1 2207.211,E2 2207.211} C_VEL
LIN {X 0,Y 575.877,Z 563.28,A -85,B 0,C 180,E1 2212.939,E2 2212.939} C_VEL
LIN {X 0,Y 575.852,Z 563.28,A -85,B 0,C 180,E1 2218.393,E2 2218.393} C_VEL
LIN {X 0,Y 575.668,Z 563.28,A -85,B 0,C 180,E1 2223.537,E2 2223.537} C_VEL
LIN {X 0,Y 575.746,Z 563.28,A -85,B 0,C 180,E1 2228.474,E2 2228.474} C_VEL
LIN {X 0,Y 575.962,Z 563.28,A -85,B 0,C 180,E1 2233.251,E2 2233.251} C_VEL
LIN {X 0,Y 575.959,Z 563.28,A -85,B 0,C 180,E1 2237.902,E2 2237.902} C_VEL
LIN {X 0,Y 576.01,Z 563.28,A -85,B 0,C 180,E1 2242.474,E2 2242.474} C_VEL
LIN {X 0,Y 576.139,Z 563.28,A -85,B 0,C 180,E1 2246.998,E2 2246.998} C_VEL
LIN {X 0,Y 576.244,Z 563.28,A -85,B 0,C 180,E1 2251.501,E2 2251.501} C_VEL
LIN {X 0,Y 576.249,Z 563.28,A -85,B 0,C 180,E1 2256.013,E2 2256.013} C_VEL
LIN {X 0,Y 575.875,Z 563.28,A -85,B 0,C 180,E1 2262.101,E2 2262.101} C_VEL
LIN {X 0,Y 575.888,Z 563.28,A -85,B 0,C 180,E1 2266.753,E2 2266.753} C_VEL
LIN {X 0,Y 575.858,Z 563.28,A -85,B 0,C 180,E1 2271.523,E2 2271.523} C_VEL
LIN {X 0,Y 575.693,Z 563.28,A -85,B 0,C 180,E1 2276.973,E2 2276.973} C_VEL
LIN {X 0,Y 575.68,Z 563.28,A -85,B 0,C 180,E1 2281.619,E2 2281.619} C_VEL
LIN {X 0,Y 575.951,Z 563.28,A -85,B 0,C 180,E1 2287.058,E2 2287.058} C_VEL
LIN {X 0,Y 575.684,Z 563.28,A -85,B 0,C 180,E1 2292.964,E2 2292.964} C_VEL
LIN {X 0,Y 575.774,Z 563.28,A -85,B 0,C 180,E1 2299.063,E2 2299.063} C_VEL
LIN {X 0,Y 575.687,Z 563.28,A -85,B 0,C 180,E1 2304.782,E2 2304.782} C_VEL
LIN {X 0,Y 575.724,Z 563.28,A -85,B 0,C 180,E1 2310.131,E2 2310.131} C_VEL
LIN {X 0,Y 575.879,Z 563.28,A -85,B 0,C 180,E1 2315.211,E2 2315.211} C_VEL
LIN {X 0,Y 576.012,Z 563.28,A -85,B 0,C 180,E1 2320.583,E2 2320.583} C_VEL
LIN {X 0,Y 575.754,Z 563.28,A -85,B 0,C 180,E1 2324.804,E2 2324.804} C_VEL
LIN {X 0,Y 575.885,Z 563.28,A -85,B 0,C 180,E1 2330.953,E2 2330.953} C_VEL
LIN {X 0,Y 575.962,Z 563.28,A -85,B 0,C 180,E1 2335.49,E2 2335.49} C_VEL
LIN {X 0,Y 576.027,Z 563.28,A -85,B 0,C 180,E1 2339.998,E2 2339.998} C_VEL
LIN {X 0,Y 575.903,Z 563.28,A -85,B 0,C 180,E1 2345.311,E2 2345.311} C_VEL
LIN {X 0,Y 575.976,Z 563.28,A -85,B 0,C 180,E1 2349.258,E2 2349.258} C_VEL
LIN {X 0,Y 571.942,Z 563.28,A -85,B 0,C 180,E1 2350.953,E2 2350.953} C_VEL
LIN {X 0,Y 568.053,Z 563.28,A -85,B 0,C 180,E1 2352.672,E2 2352.672} C_VEL
LIN {X 0,Y 568.034,Z 563.28,A -85,B 0,C 180,E1 2358.588,E2 2358.588} C_VEL
LIN {X 0,Y 567.928,Z 563.28,A -85,B 0,C 180,E1 2363.486,E2 2363.486} C_VEL
LIN {X 0,Y 567.857,Z 563.28,A -85,B 0,C 180,E1 2368.724,E2 2368.724} C_VEL
LIN {X 0,Y 567.987,Z 563.28,A -85,B 0,C 180,E1 2374.552,E2 2374.552} C_VEL
LIN {X 0,Y 567.812,Z 563.28,A -85,B 0,C 180,E1 2379.627,E2 2379.627} C_VEL
LIN {X 0,Y 567.653,Z 563.28,A -85,B 0,C 180,E1 2385.866,E2 2385.866} C_VEL
LIN {X 0,Y 567.808,Z 563.28,A -85,B 0,C 180,E1 2390.414,E2 2390.414} C_VEL
LIN {X 0,Y 568.036,Z 563.28,A -85,B 0,C 180,E1 2396.09,E2 2396.09} C_VEL
LIN {X 0,Y 568.095,Z 563.28,A -85,B 0,C 180,E1 2398.3,E2 2398.3} C_VEL
LIN {X 0,Y 574.029,Z 578.99,A -85,B 0,C 180,E1 2398.899,E2 2398.899} C_VEL
LIN {X 0,Y 573.947,Z 627.071,A -85,B 0,C 180,E1 2399.764,E2 2399.764} C_VEL
LIN {X 0,Y 573.212,Z 665.775,A -85,B 0,C 180,E1 2401.067,E2 2401.067} C_VEL
LIN {X 0,Y 572.185,Z 703.317,A -85,B 0,C 180,E1 2402.966,E2 2402.966} C_VEL
LIN {X 0,Y 571.092,Z 738.03,A -85,B 0,C 180,E1 2405.393,E2 2405.393} C_VEL
LIN {X 0,Y 570.101,Z 768.964,A -85,B 0,C 180,E1 2408.249,E2 2408.249} C_VEL
LIN {X 0,Y 569.283,Z 796.934,A -85,B 0,C 180,E1 2411.62,E2 2411.62} C_VEL
LIN {X 0,Y 568.735,Z 820.193,A -85,B 0,C 180,E1 2415.342,E2 2415.342} C_VEL
LIN {X 0,Y 568.495,Z 838.031,A -85,B 0,C 180,E1 2419.291,E2 2419.291} C_VEL
LIN {X 0,Y 568.366,Z 849.585,A -85,B 0,C 180,E1 2423.137,E2 2423.137} C_VEL
LIN {X 0,Y 568.356,Z 855.92,A -85,B 0,C 180,E1 2426.955,E2 2426.955} C_VEL
LIN {X 0,Y 568.268,Z 857.5,A -85,B 0,C 180,E1 2429.999,E2 2429.999} C_VEL
LIN {X 0,Y 568.228,Z 855.922,A -85,B 0,C 180,E1 2433.044,E2 2433.044} C_VEL
LIN {X 0,Y 568.294,Z 849.589,A -85,B 0,C 180,E1 2436.862,E2 2436.862} C_VEL
LIN {X 0,Y 568.386,Z 837.686,A -85,B 0,C 180,E1 2440.806,E2 2440.806} C_VEL
LIN {X 0,Y 568.737,Z 820.248,A -85,B 0,C 180,E1 2444.648,E2 2444.648} C_VEL
LIN {X 0,Y 569.292,Z 796.963,A -85,B 0,C 180,E1 2448.376,E2 2448.376} C_VEL
LIN {X 0,Y 570.08,Z 768.978,A -85,B 0,C 180,E1 2451.751,E2 2451.751} C_VEL
LIN {X 0,Y 571.084,Z 736.861,A -85,B 0,C 180,E1 2454.704,E2 2454.704} C_VEL
LIN {X 0,Y 572.222,Z 700.515,A -85,B 0,C 180,E1 2457.206,E2 2457.206} C_VEL
LIN {X 0,Y 573.242,Z 660.348,A -85,B 0,C 180,E1 2459.163,E2 2459.163} C_VEL
LIN {X 0,Y 574.021,Z 620.37,A -85,B 0,C 180,E1 2460.396,E2 2460.396} C_VEL
LIN {X 0,Y 573.63,Z 576.618,A -85,B 0,C 180,E1 2461.16,E2 2461.16} C_VEL
LIN {X 0,Y 567.889,Z 563.28,A -85,B 0,C 180,E1 2461.759,E2 2461.759} C_VEL
LIN {X 0,Y 567.983,Z 563.28,A -85,B 0,C 180,E1 2467.665,E2 2467.665} C_VEL
LIN {X 0,Y 567.718,Z 563.28,A -85,B 0,C 180,E1 2474.141,E2 2474.141} C_VEL
LIN {X 0,Y 567.817,Z 563.28,A -85,B 0,C 180,E1 2478.367,E2 2478.367} C_VEL
LIN {X 0,Y 567.806,Z 563.28,A -85,B 0,C 180,E1 2484.223,E2 2484.223} C_VEL
LIN {X 0,Y 567.796,Z 563.28,A -85,B 0,C 180,E1 2489.674,E2 2489.674} C_VEL
LIN {X 0,Y 567.913,Z 563.28,A -85,B 0,C 180,E1 2494.843,E2 2494.843} C_VEL
LIN {X 0,Y 567.996,Z 563.28,A -85,B 0,C 180,E1 2499.797,E2 2499.797} C_VEL
LIN {X 0,Y 567.872,Z 563.28,A -85,B 0,C 180,E1 2504.592,E2 2504.592} C_VEL
LIN {X 0,Y 567.97,Z 563.28,A -85,B 0,C 180,E1 2510.829,E2 2510.829} C_VEL
LIN {X 0,Y 568.051,Z 563.28,A -85,B 0,C 180,E1 2515.431,E2 2515.431} C_VEL
LIN {X 0,Y 568.13,Z 563.28,A -85,B 0,C 180,E1 2520.002,E2 2520.002} C_VEL
LIN {X 0,Y 568.106,Z 563.28,A -85,B 0,C 180,E1 2524.572,E2 2524.572} C_VEL
LIN {X 0,Y 568.08,Z 563.28,A -85,B 0,C 180,E1 2529.172,E2 2529.172} C_VEL
LIN {X 0,Y 568.115,Z 563.28,A -85,B 0,C 180,E1 2533.832,E2 2533.832} C_VEL
LIN {X 0,Y 568.058,Z 563.28,A -85,B 0,C 180,E1 2538.59,E2 2538.59} C_VEL
LIN {X 0,Y 567.935,Z 563.28,A -85,B 0,C 180,E1 2543.489,E2 2543.489} C_VEL
LIN {X 0,Y 567.863,Z 563.28,A -85,B 0,C 180,E1 2548.728,E2 2548.728} C_VEL
LIN {X 0,Y 567.983,Z 563.28,A -85,B 0,C 180,E1 2554.554,E2 2554.554} C_VEL
LIN {X 0,Y 567.832,Z 563.28,A -85,B 0,C 180,E1 2559.629,E2 2559.629} C_VEL
LIN {X 0,Y 567.67,Z 563.28,A -85,B 0,C 180,E1 2564.134,E2 2564.134} C_VEL
LIN {X 0,Y 567.797,Z 563.28,A -85,B 0,C 180,E1 2568.364,E2 2568.364} C_VEL
LIN {X 0,Y 567.995,Z 563.28,A -85,B 0,C 180,E1 2574.235,E2 2574.235} C_VEL
LIN {X 0,Y 567.927,Z 563.28,A -85,B 0,C 180,E1 2579.68,E2 2579.68} C_VEL
LIN {X 0,Y 567.775,Z 563.28,A -85,B 0,C 180,E1 2584.835,E2 2584.835} C_VEL
LIN {X 0,Y 567.82,Z 563.28,A -85,B 0,C 180,E1 2589.79,E2 2589.79} C_VEL
LIN {X 0,Y 567.918,Z 563.28,A -85,B 0,C 180,E1 2594.592,E2 2594.592} C_VEL
LIN {X 0,Y 567.968,Z 563.28,A -85,B 0,C 180,E1 2599.435,E2 2599.435} C_VEL
LIN {X 0,Y 568.013,Z 563.28,A -85,B 0,C 180,E1 2603.901,E2 2603.901} C_VEL
LIN {X 0,Y 567.989,Z 563.28,A -85,B 0,C 180,E1 2608.478,E2 2608.478} C_VEL
LIN {X 0,Y 568.051,Z 563.28,A -85,B 0,C 180,E1 2613.046,E2 2613.046} C_VEL
LIN {X 0,Y 567.981,Z 563.28,A -85,B 0,C 180,E1 2617.634,E2 2617.634} C_VEL
LIN {X 0,Y 567.962,Z 563.28,A -85,B 0,C 180,E1 2622.273,E2 2622.273} C_VEL
LIN {X 0,Y 567.958,Z 563.28,A -85,B 0,C 180,E1 2626.994,E2 2626.994} C_VEL
LIN {X 0,Y 567.908,Z 563.28,A -85,B 0,C 180,E1 2631.84,E2 2631.84} C_VEL
LIN {X 0,Y 567.807,Z 563.28,A -85,B 0,C 180,E1 2636.86,E2 2636.86} C_VEL
LIN {X 0,Y 567.74,Z 563.28,A -85,B 0,C 180,E1 2642.113,E2 2642.113} C_VEL
LIN {X 0,Y 568.026,Z 563.28,A -85,B 0,C 180,E1 2647.664,E2 2647.664} C_VEL
LIN {X 0,Y 567.747,Z 563.28,A -85,B 0,C 180,E1 2654.139,E2 2654.139} C_VEL
LIN {X 0,Y 567.828,Z 563.28,A -85,B 0,C 180,E1 2660.371,E2 2660.371} C_VEL
LIN {X 0,Y 567.694,Z 563.28,A -85,B 0,C 180,E1 2665.491,E2 2665.491} C_VEL
LIN {X 0,Y 567.764,Z 563.28,A -85,B 0,C 180,E1 2671.293,E2 2671.293} C_VEL
LIN {X 0,Y 567.844,Z 563.28,A -85,B 0,C 180,E1 2676.507,E2 2676.507} C_VEL
LIN {X 0,Y 568.092,Z 563.28,A -85,B 0,C 180,E1 2681.411,E2 2681.411} C_VEL
LIN {X 0,Y 567.771,Z 563.28,A -85,B 0,C 180,E1 2687.722,E2 2687.722} C_VEL
LIN {X 0,Y 568.043,Z 563.28,A -85,B 0,C 180,E1 2692.879,E2 2692.879} C_VEL
LIN {X 0,Y 568.372,Z 563.28,A -85,B 0,C 180,E1 2698.477,E2 2698.477} C_VEL
LIN {X 0,Y 568.095,Z 563.28,A -85,B 0,C 180,E1 2704.569,E2 2704.569} C_VEL
LIN {X 0,Y 568.08,Z 563.28,A -85,B 0,C 180,E1 2709.242,E2 2709.242} C_VEL
LIN {X 0,Y 568.053,Z 563.28,A -85,B 0,C 180,E1 2712.672,E2 2712.672} C_VEL
LIN {X 0,Y 565.468,Z 563.28,A -85,B 0,C 180,E1 2713.97,E2 2713.97} C_VEL
LIN {X 0,Y 560.06,Z 563.28,A -85,B 0,C 180,E1 2715.912,E2 2715.912} C_VEL
LIN {X 0,Y 559.968,Z 563.28,A -85,B 0,C 180,E1 2716.136,E2 2716.136} C_VEL
LIN {X 0,Y 559.997,Z 563.28,A -85,B 0,C 180,E1 2720.504,E2 2720.504} C_VEL
LIN {X 0,Y 559.865,Z 563.28,A -85,B 0,C 180,E1 2725.545,E2 2725.545} C_VEL
LIN {X 0,Y 559.935,Z 563.28,A -85,B 0,C 180,E1 2730.798,E2 2730.798} C_VEL
LIN {X 0,Y 560.047,Z 563.28,A -85,B 0,C 180,E1 2736.351,E2 2736.351} C_VEL
LIN {X 0,Y 559.788,Z 563.28,A -85,B 0,C 180,E1 2742.367,E2 2742.367} C_VEL
LIN {X 0,Y 559.825,Z 563.28,A -85,B 0,C 180,E1 2747.632,E2 2747.632} C_VEL
LIN {X 0,Y 560.052,Z 563.28,A -85,B 0,C 180,E1 2753.928,E2 2753.928} C_VEL
LIN {X 0,Y 560.171,Z 563.28,A -85,B 0,C 180,E1 2757.793,E2 2757.793} C_VEL
LIN {X 0,Y 567.354,Z 582.005,A -85,B 0,C 180,E1 2758.535,E2 2758.535} C_VEL
LIN {X 0,Y 567.089,Z 627.973,A -85,B 0,C 180,E1 2759.384,E2 2759.384} C_VEL
LIN {X 0,Y 566.202,Z 666.662,A -85,B 0,C 180,E1 2760.713,E2 2760.713} C_VEL
LIN {X 0,Y 565.011,Z 703.225,A -85,B 0,C 180,E1 2762.588,E2 2762.588} C_VEL
LIN {X 0,Y 563.711,Z 738.227,A -85,B 0,C 180,E1 2765.065,E2 2765.065} C_VEL
LIN {X 0,Y 562.533,Z 768.967,A -85,B 0,C 180,E1 2767.941,E2 2767.941} C_VEL
LIN {X 0,Y 561.576,Z 796.801,A -85,B 0,C 180,E1 2771.34,E2 2771.34} C_VEL
LIN {X 0,Y 560.932,Z 819.773,A -85,B 0,C 180,E1 2775.055,E2 2775.055} C_VEL
LIN {X 0,Y 560.557,Z 836.529,A -85,B 0,C 180,E1 2778.745,E2 2778.745} C_VEL
LIN {X 0,Y 560.423,Z 847.682,A -85,B 0,C 180,E1 2782.262,E2 2782.262} C_VEL
LIN {X 0,Y 560.317,Z 853.973,A -85,B 0,C 180,E1 2785.365,E2 2785.365} C_VEL
LIN {X 0,Y 560.364,Z 857.097,A -85,B 0,C 180,E1 2788.456,E2 2788.456} C_VEL
LIN {X 0,Y 560.487,Z 857.098,A -85,B 0,C 180,E1 2791.542,E2 2791.542} C_VEL
LIN {X 0,Y 560.488,Z 852.799,A -85,B 0,C 180,E1 2795.373,E2 2795.373} C_VEL
LIN {X 0,Y 560.511,Z 843.295,A -85,B 0,C 180,E1 2799.295,E2 2799.295} C_VEL
LIN {X 0,Y 560.779,Z 828.3,A -85,B 0,C 180,E1 2803.221,E2 2803.221} C_VEL
LIN {X 0,Y 561.215,Z 807.921,A -85,B 0,C 180,E1 2807.002,E2 2807.002} C_VEL
LIN {X 0,Y 562.061,Z 781.617,A -85,B 0,C 180,E1 2810.632,E2 2810.632} C_VEL
LIN {X 0,Y 563.175,Z 750.978,A -85,B 0,C 180,E1 2813.833,E2 2813.833} C_VEL
LIN {X 0,Y 564.47,Z 716.608,A -85,B 0,C 180,E1 2816.554,E2 2816.554} C_VEL
LIN {X 0,Y 565.787,Z 679.73,A -85,B 0,C 180,E1 2818.69,E2 2818.69} C_VEL
LIN {X 0,Y 566.8,Z 642.887,A -85,B 0,C 180,E1 2820.179,E2 2820.179} C_VEL
LIN {X 0,Y 567.483,Z 606.501,A -85,B 0,C 180,E1 2821.076,E2 2821.076} C_VEL
LIN {X 0,Y 566.646,Z 578.829,A -85,B 0,C 180,E1 2821.555,E2 2821.555} C_VEL
LIN {X 0,Y 559.931,Z 563.28,A -85,B 0,C 180,E1 2822.223,E2 2822.223} C_VEL
LIN {X 0,Y 559.968,Z 563.28,A -85,B 0,C 180,E1 2828.301,E2 2828.301} C_VEL
LIN {X 0,Y 559.789,Z 563.28,A -85,B 0,C 180,E1 2834.496,E2 2834.496} C_VEL
LIN {X 0,Y 559.836,Z 563.28,A -85,B 0,C 180,E1 2839.694,E2 2839.694} C_VEL
LIN {X 0,Y 559.793,Z 563.28,A -85,B 0,C 180,E1 2845.525,E2 2845.525} C_VEL
LIN {X 0,Y 559.833,Z 563.28,A -85,B 0,C 180,E1 2850.978,E2 2850.978} C_VEL
LIN {X 0,Y 559.935,Z 563.28,A -85,B 0,C 180,E1 2856.388,E2 2856.388} C_VEL
LIN {X 0,Y 560.109,Z 563.28,A -85,B 0,C 180,E1 2861.14,E2 2861.14} C_VEL
LIN {X 0,Y 559.791,Z 563.28,A -85,B 0,C 180,E1 2866.031,E2 2866.031} C_VEL
LIN {X 0,Y 560.065,Z 563.28,A -85,B 0,C 180,E1 2870.698,E2 2870.698} C_VEL
LIN {X 0,Y 560.157,Z 563.28,A -85,B 0,C 180,E1 2875.366,E2 2875.366} C_VEL
LIN {X 0,Y 560.229,Z 563.28,A -85,B 0,C 180,E1 2880.002,E2 2880.002} C_VEL
LIN {X 0,Y 560.188,Z 563.28,A -85,B 0,C 180,E1 2884.672,E2 2884.672} C_VEL
LIN {X 0,Y 560.166,Z 563.28,A -85,B 0,C 180,E1 2889.303,E2 2889.303} C_VEL
LIN {X 0,Y 560.146,Z 563.28,A -85,B 0,C 180,E1 2894.114,E2 2894.114} C_VEL
LIN {X 0,Y 560.046,Z 563.28,A -85,B 0,C 180,E1 2899.431,E2 2899.431} C_VEL
LIN {X 0,Y 559.976,Z 563.28,A -85,B 0,C 180,E1 2903.843,E2 2903.843} C_VEL
LIN {X 0,Y 559.931,Z 563.28,A -85,B 0,C 180,E1 2909.02,E2 2909.02} C_VEL
LIN {X 0,Y 560.093,Z 563.28,A -85,B 0,C 180,E1 2914.458,E2 2914.458} C_VEL
LIN {X 0,Y 559.85,Z 563.28,A -85,B 0,C 180,E1 2920.309,E2 2920.309} C_VEL
LIN {X 0,Y 559.729,Z 563.28,A -85,B 0,C 180,E1 2925.498,E2 2925.498} C_VEL
LIN {X 0,Y 559.9,Z 563.28,A -85,B 0,C 180,E1 2931.408,E2 2931.408} C_VEL
LIN {X 0,Y 560.038,Z 563.28,A -85,B 0,C 180,E1 2936.647,E2 2936.647} C_VEL
LIN {X 0,Y 559.953,Z 563.28,A -85,B 0,C 180,E1 2940.983,E2 2940.983} C_VEL
LIN {X 0,Y 559.941,Z 563.28,A -85,B 0,C 180,E1 2946.39,E2 2946.39} C_VEL
LIN {X 0,Y 560.111,Z 563.28,A -85,B 0,C 180,E1 2952.762,E2 2952.762} C_VEL
LIN {X 0,Y 560.161,Z 563.28,A -85,B 0,C 180,E1 2957.555,E2 2957.555} C_VEL
LIN {X 0,Y 560.219,Z 563.28,A -85,B 0,C 180,E1 2962.261,E2 2962.261} C_VEL
LIN {X 0,Y 560.322,Z 563.28,A -85,B 0,C 180,E1 2966.913,E2 2966.913} C_VEL
LIN {X 0,Y 560.448,Z 563.28,A -85,B 0,C 180,E1 2971.544,E2 2971.544} C_VEL
LIN {X 0,Y 560.395,Z 563.28,A -85,B 0,C 180,E1 2976.184,E2 2976.184} C_VEL
LIN {X 0,Y 560.039,Z 563.28,A -85,B 0,C 180,E1 2982.449,E2 2982.449} C_VEL
LIN {X 0,Y 560.024,Z 563.28,A -85,B 0,C 180,E1 2987.242,E2 2987.242} C_VEL
LIN {X 0,Y 559.956,Z 563.28,A -85,B 0,C 180,E1 2992.166,E2 2992.166} C_VEL
LIN {X 0,Y 559.84,Z 563.28,A -85,B 0,C 180,E1 2997.273,E2 2997.273} C_VEL
LIN {X 0,Y 559.769,Z 563.28,A -85,B 0,C 180,E1 3002.627,E2 3002.627} C_VEL
LIN {X 0,Y 560.009,Z 563.28,A -85,B 0,C 180,E1 3008.3,E2 3008.3} C_VEL
LIN {X 0,Y 559.815,Z 563.28,A -85,B 0,C 180,E1 3014.496,E2 3014.496} C_VEL
LIN {X 0,Y 559.847,Z 563.28,A -85,B 0,C 180,E1 3019.691,E2 3019.691} C_VEL
LIN {X 0,Y 559.816,Z 563.28,A -85,B 0,C 180,E1 3025.522,E2 3025.522} C_VEL
LIN {X 0,Y 559.849,Z 563.28,A -85,B 0,C 180,E1 3030.975,E2 3030.975} C_VEL
LIN {X 0,Y 559.935,Z 563.28,A -85,B 0,C 180,E1 3036.391,E2 3036.391} C_VEL
LIN {X 0,Y 560.148,Z 563.28,A -85,B 0,C 180,E1 3041.138,E2 3041.138} C_VEL
LIN {X 0,Y 559.798,Z 563.28,A -85,B 0,C 180,E1 3046.034,E2 3046.034} C_VEL
LIN {X 0,Y 560.072,Z 563.28,A -85,B 0,C 180,E1 3050.695,E2 3050.695} C_VEL
LIN {X 0,Y 560.174,Z 563.28,A -85,B 0,C 180,E1 3055.363,E2 3055.363} C_VEL
LIN {X 0,Y 560.25,Z 563.28,A -85,B 0,C 180,E1 3059.998,E2 3059.998} C_VEL
LIN {X 0,Y 560.199,Z 563.28,A -85,B 0,C 180,E1 3064.669,E2 3064.669} C_VEL
LIN {X 0,Y 560.181,Z 563.28,A -85,B 0,C 180,E1 3069.3,E2 3069.3} C_VEL
LIN {X 0,Y 560.171,Z 563.28,A -85,B 0,C 180,E1 3074.118,E2 3074.118} C_VEL
LIN {X 0,Y 559.968,Z 563.28,A -85,B 0,C 180,E1 3076.136,E2 3076.136} C_VEL
LIN {X 0,Y 556.087,Z 563.28,A -85,B 0,C 180,E1 3077.882,E2 3077.882} C_VEL
LIN {X 0,Y 552.082,Z 563.28,A -85,B 0,C 180,E1 3079.652,E2 3079.652} C_VEL
LIN {X 0,Y 551.971,Z 563.28,A -85,B 0,C 180,E1 3085.553,E2 3085.553} C_VEL
LIN {X 0,Y 552.007,Z 563.28,A -85,B 0,C 180,E1 3091.289,E2 3091.289} C_VEL
LIN {X 0,Y 552.036,Z 563.28,A -85,B 0,C 180,E1 3096.966,E2 3096.966} C_VEL
LIN {X 0,Y 551.824,Z 563.28,A -85,B 0,C 180,E1 3103.126,E2 3103.126} C_VEL
LIN {X 0,Y 551.952,Z 563.28,A -85,B 0,C 180,E1 3108.992,E2 3108.992} C_VEL
LIN {X 0,Y 552.147,Z 563.28,A -85,B 0,C 180,E1 3115.07,E2 3115.07} C_VEL
LIN {X 0,Y 552.215,Z 563.28,A -85,B 0,C 180,E1 3117.271,E2 3117.271} C_VEL
LIN {X 0,Y 560.653,Z 583.884,A -85,B 0,C 180,E1 3118.143,E2 3118.143} C_VEL
LIN {X 0,Y 560.281,Z 627.99,A -85,B 0,C 180,E1 3118.971,E2 3118.971} C_VEL
LIN {X 0,Y 559.251,Z 665.629,A -85,B 0,C 180,E1 3120.267,E2 3120.267} C_VEL
LIN {X 0,Y 557.895,Z 702.358,A -85,B 0,C 180,E1 3122.151,E2 3122.151} C_VEL
LIN {X 0,Y 556.382,Z 737.371,A -85,B 0,C 180,E1 3124.642,E2 3124.642} C_VEL
LIN {X 0,Y 554.977,Z 768.97,A -85,B 0,C 180,E1 3127.624,E2 3127.624} C_VEL
LIN {X 0,Y 553.832,Z 797.173,A -85,B 0,C 180,E1 3131.121,E2 3131.121} C_VEL
LIN {X 0,Y 553.084,Z 819.417,A -85,B 0,C 180,E1 3134.77,E2 3134.77} C_VEL
LIN {X 0,Y 552.67,Z 836.532,A -85,B 0,C 180,E1 3138.582,E2 3138.582} C_VEL
LIN {X 0,Y 552.534,Z 847.682,A -85,B 0,C 180,E1 3142.151,E2 3142.151} C_VEL
LIN {X 0,Y 552.447,Z 853.976,A -85,B 0,C 180,E1 3145.299,E2 3145.299} C_VEL
LIN {X 0,Y 552.468,Z 857.099,A -85,B 0,C 180,E1 3148.434,E2 3148.434} C_VEL
LIN {X 0,Y 552.581,Z 857.1,A -85,B 0,C 180,E1 3151.564,E2 3151.564} C_VEL
LIN {X 0,Y 552.548,Z 852.354,A -85,B 0,C 180,E1 3155.693,E2 3155.693} C_VEL
LIN {X 0,Y 552.613,Z 843.294,A -85,B 0,C 180,E1 3159.429,E2 3159.429} C_VEL
LIN {X 0,Y 552.925,Z 828.298,A -85,B 0,C 180,E1 3163.413,E2 3163.413} C_VEL
LIN {X 0,Y 553.482,Z 806.946,A -85,B 0,C 180,E1 3167.409,E2 3167.409} C_VEL
LIN {X 0,Y 554.511,Z 779.91,A -85,B 0,C 180,E1 3171.135,E2 3171.135} C_VEL
LIN {X 0,Y 555.811,Z 749.507,A -85,B 0,C 180,E1 3174.307,E2 3174.307} C_VEL
LIN {X 0,Y 557.295,Z 715.023,A -85,B 0,C 180,E1 3177.038,E2 3177.038} C_VEL
LIN {X 0,Y 558.871,Z 676.453,A -85,B 0,C 180,E1 3179.249,E2 3179.249} C_VEL
LIN {X 0,Y 559.982,Z 639.396,A -85,B 0,C 180,E1 3180.702,E2 3180.702} C_VEL
LIN {X 0,Y 560.77,Z 599.358,A -85,B 0,C 180,E1 3181.616,E2 3181.616} C_VEL
LIN {X 0,Y 559.88,Z 581.246,A -85,B 0,C 180,E1 3181.946,E2 3181.946} C_VEL
LIN {X 0,Y 551.95,Z 563.28,A -85,B 0,C 180,E1 3182.796,E2 3182.796} C_VEL
LIN {X 0,Y 551.993,Z 563.28,A -85,B 0,C 180,E1 3188.958,E2 3188.958} C_VEL
LIN {X 0,Y 551.912,Z 563.28,A -85,B 0,C 180,E1 3195.305,E2 3195.305} C_VEL
LIN {X 0,Y 551.943,Z 563.28,A -85,B 0,C 180,E1 3201.04,E2 3201.04} C_VEL
LIN {X 0,Y 551.841,Z 563.28,A -85,B 0,C 180,E1 3206.848,E2 3206.848} C_VEL
LIN {X 0,Y 551.925,Z 563.28,A -85,B 0,C 180,E1 3212.305,E2 3212.305} C_VEL
LIN {X 0,Y 552.003,Z 563.28,A -85,B 0,C 180,E1 3217.5,E2 3217.5} C_VEL
LIN {X 0,Y 552.214,Z 563.28,A -85,B 0,C 180,E1 3223.022,E2 3223.022} C_VEL
LIN {X 0,Y 552.174,Z 563.28,A -85,B 0,C 180,E1 3229.677,E2 3229.677} C_VEL
LIN {X 0,Y 552.259,Z 563.28,A -85,B 0,C 180,E1 3235.3,E2 3235.3} C_VEL
LIN {X 0,Y 552.331,Z 563.28,A -85,B 0,C 180,E1 3240.002,E2 3240.002} C_VEL
LIN {X 0,Y 552.31,Z 563.28,A -85,B 0,C 180,E1 3244.703,E2 3244.703} C_VEL
LIN {X 0,Y 552.14,Z 563.28,A -85,B 0,C 180,E1 3250.303,E2 3250.303} C_VEL
LIN {X 0,Y 552.104,Z 563.28,A -85,B 0,C 180,E1 3255.863,E2 3255.863} C_VEL
LIN {X 0,Y 552.068,Z 563.28,A -85,B 0,C 180,E1 3261.669,E2 3261.669} C_VEL
LIN {X 0,Y 551.993,Z 563.28,A -85,B 0,C 180,E1 3267.695,E2 3267.695} C_VEL
LIN {X 0,Y 552.154,Z 563.28,A -85,B 0,C 180,E1 3273.135,E2 3273.135} C_VEL
LIN {X 0,Y 551.973,Z 563.28,A -85,B 0,C 180,E1 3278.962,E2 3278.962} C_VEL
LIN {X 0,Y 551.833,Z 563.28,A -85,B 0,C 180,E1 3284.686,E2 3284.686} C_VEL
LIN {X 0,Y 551.932,Z 563.28,A -85,B 0,C 180,E1 3289.956,E2 3289.956} C_VEL
LIN {X 0,Y 552.162,Z 563.28,A -85,B 0,C 180,E1 3295.074,E2 3295.074} C_VEL
LIN {X 0,Y 552.065,Z 563.28,A -85,B 0,C 180,E1 3301.009,E2 3301.009} C_VEL
LIN {X 0,Y 551.972,Z 563.28,A -85,B 0,C 180,E1 3305.791,E2 3305.791} C_VEL
LIN {X 0,Y 552.127,Z 563.28,A -85,B 0,C 180,E1 3310.855,E2 3310.855} C_VEL
LIN {X 0,Y 552.248,Z 563.28,A -85,B 0,C 180,E1 3315.764,E2 3315.764} C_VEL
LIN {X 0,Y 552.304,Z 563.28,A -85,B 0,C 180,E1 3322.149,E2 3322.149} C_VEL
LIN {X 0,Y 552.422,Z 563.28,A -85,B 0,C 180,E1 3326.869,E2 3326.869} C_VEL
LIN {X 0,Y 552.541,Z 563.28,A -85,B 0,C 180,E1 3331.566,E2 3331.566} C_VEL
LIN {X 0,Y 552.463,Z 563.28,A -85,B 0,C 180,E1 3336.273,E2 3336.273} C_VEL
LIN {X 0,Y 552.127,Z 563.28,A -85,B 0,C 180,E1 3342.63,E2 3342.63} C_VEL
LIN {X 0,Y 552.113,Z 563.28,A -85,B 0,C 180,E1 3347.497,E2 3347.497} C_VEL
LIN {X 0,Y 552.025,Z 563.28,A -85,B 0,C 180,E1 3352.502,E2 3352.502} C_VEL
LIN {X 0,Y 551.886,Z 563.28,A -85,B 0,C 180,E1 3357.7,E2 3357.7} C_VEL
LIN {X 0,Y 551.863,Z 563.28,A -85,B 0,C 180,E1 3363.154,E2 3363.154} C_VEL
LIN {X 0,Y 552.03,Z 563.28,A -85,B 0,C 180,E1 3368.957,E2 3368.957} C_VEL
LIN {X 0,Y 551.934,Z 563.28,A -85,B 0,C 180,E1 3375.305,E2 3375.305} C_VEL
LIN {X 0,Y 551.958,Z 563.28,A -85,B 0,C 180,E1 3381.037,E2 3381.037} C_VEL
LIN {X 0,Y 551.86,Z 563.28,A -85,B 0,C 180,E1 3386.845,E2 3386.845} C_VEL
LIN {X 0,Y 551.945,Z 563.28,A -85,B 0,C 180,E1 3392.303,E2 3392.303} C_VEL
LIN {X 0,Y 552.024,Z 563.28,A -85,B 0,C 180,E1 3397.497,E2 3397.497} C_VEL
LIN {X 0,Y 552.212,Z 563.28,A -85,B 0,C 180,E1 3403.027,E2 3403.027} C_VEL
LIN {X 0,Y 552.136,Z 563.28,A -85,B 0,C 180,E1 3409.707,E2 3409.707} C_VEL
LIN {X 0,Y 552.276,Z 563.28,A -85,B 0,C 180,E1 3415.297,E2 3415.297} C_VEL
LIN {X 0,Y 552.352,Z 563.28,A -85,B 0,C 180,E1 3419.998,E2 3419.998} C_VEL
LIN {X 0,Y 552.321,Z 563.28,A -85,B 0,C 180,E1 3424.7,E2 3424.7} C_VEL
LIN {X 0,Y 552.156,Z 563.28,A -85,B 0,C 180,E1 3430.304,E2 3430.304} C_VEL
LIN {X 0,Y 552.074,Z 563.28,A -85,B 0,C 180,E1 3435.861,E2 3435.861} C_VEL
LIN {X 0,Y 552.082,Z 563.28,A -85,B 0,C 180,E1 3439.652,E2 3439.652} C_VEL
LIN {X 0,Y 548.061,Z 563.28,A -85,B 0,C 180,E1 3441.421,E2 3441.421} C_VEL
LIN {X 0,Y 544.082,Z 563.28,A -85,B 0,C 180,E1 3443.215,E2 3443.215} C_VEL
LIN {X 0,Y 544.061,Z 563.28,A -85,B 0,C 180,E1 3448.13,E2 3448.13} C_VEL
LIN {X 0,Y 544.22,Z 563.28,A -85,B 0,C 180,E1 3453.711,E2 3453.711} C_VEL
LIN {X 0,Y 544.006,Z 563.28,A -85,B 0,C 180,E1 3459.639,E2 3459.639} C_VEL
LIN {X 0,Y 543.921,Z 563.28,A -85,B 0,C 180,E1 3466.16,E2 3466.16} C_VEL
LIN {X 0,Y 544.112,Z 563.28,A -85,B 0,C 180,E1 3472.4,E2 3472.4} C_VEL
LIN {X 0,Y 544.295,Z 563.28,A -85,B 0,C 180,E1 3476.736,E2 3476.736} C_VEL
LIN {X 0,Y 554.005,Z 587.061,A -85,B 0,C 180,E1 3477.762,E2 3477.762} C_VEL
LIN {X 0,Y 553.447,Z 629.767,A -85,B 0,C 180,E1 3478.596,E2 3478.596} C_VEL
LIN {X 0,Y 552.269,Z 667.347,A -85,B 0,C 180,E1 3479.932,E2 3479.932} C_VEL
LIN {X 0,Y 550.728,Z 703.456,A -85,B 0,C 180,E1 3481.829,E2 3481.829} C_VEL
LIN {X 0,Y 548.998,Z 738.619,A -85,B 0,C 180,E1 3484.383,E2 3484.383} C_VEL
LIN {X 0,Y 547.392,Z 770.056,A -85,B 0,C 180,E1 3487.418,E2 3487.418} C_VEL
LIN {X 0,Y 546.119,Z 798.635,A -85,B 0,C 180,E1 3491.054,E2 3491.054} C_VEL
LIN {X 0,Y 545.285,Z 821.545,A -85,B 0,C 180,E1 3494.962,E2 3494.962} C_VEL
LIN {X 0,Y 544.825,Z 838.021,A -85,B 0,C 180,E1 3498.82,E2 3498.82} C_VEL
LIN {X 0,Y 544.706,Z 849.577,A -85,B 0,C 180,E1 3502.838,E2 3502.838} C_VEL
LIN {X 0,Y 544.654,Z 855.928,A -85,B 0,C 180,E1 3506.823,E2 3506.823} C_VEL
LIN {X 0,Y 544.568,Z 857.5,A -85,B 0,C 180,E1 3509.999,E2 3509.999} C_VEL
LIN {X 0,Y 544.583,Z 854.955,A -85,B 0,C 180,E1 3514.056,E2 3514.056} C_VEL
LIN {X 0,Y 544.779,Z 846.722,A -85,B 0,C 180,E1 3518.361,E2 3518.361} C_VEL
LIN {X 0,Y 545.054,Z 831.798,A -85,B 0,C 180,E1 3522.795,E2 3522.795} C_VEL
LIN {X 0,Y 545.634,Z 812.071,A -85,B 0,C 180,E1 3526.789,E2 3526.789} C_VEL
LIN {X 0,Y 546.598,Z 787.663,A -85,B 0,C 180,E1 3530.463,E2 3530.463} C_VEL
LIN {X 0,Y 548.005,Z 757.876,A -85,B 0,C 180,E1 3533.855,E2 3533.855} C_VEL
LIN {X 0,Y 549.694,Z 724.64,A -85,B 0,C 180,E1 3536.725,E2 3536.725} C_VEL
LIN {X 0,Y 551.466,Z 687.951,A -85,B 0,C 180,E1 3539.07,E2 3539.07} C_VEL
LIN {X 0,Y 552.86,Z 650.497,A -85,B 0,C 180,E1 3540.742,E2 3540.742} C_VEL
LIN {X 0,Y 553.869,Z 613.312,A -85,B 0,C 180,E1 3541.796,E2 3541.796} C_VEL
LIN {X 0,Y 553.468,Z 584.542,A -85,B 0,C 180,E1 3542.311,E2 3542.311} C_VEL
LIN {X 0,Y 544.043,Z 563.28,A -85,B 0,C 180,E1 3543.307,E2 3543.307} C_VEL
LIN {X 0,Y 544.078,Z 563.28,A -85,B 0,C 180,E1 3549.055,E2 3549.055} C_VEL
LIN {X 0,Y 543.926,Z 563.28,A -85,B 0,C 180,E1 3553.913,E2 3553.913} C_VEL
LIN {X 0,Y 544.042,Z 563.28,A -85,B 0,C 180,E1 3558.494,E2 3558.494} C_VEL
LIN {X 0,Y 543.947,Z 563.28,A -85,B 0,C 180,E1 3564.371,E2 3564.371} C_VEL
LIN {X 0,Y 543.962,Z 563.28,A -85,B 0,C 180,E1 3570.046,E2 3570.046} C_VEL
LIN {X 0,Y 544.098,Z 563.28,A -85,B 0,C 180,E1 3575.419,E2 3575.419} C_VEL
LIN {X 0,Y 544.267,Z 563.28,A -85,B 0,C 180,E1 3580.569,E2 3580.569} C_VEL
LIN {X 0,Y 543.972,Z 563.28,A -85,B 0,C 180,E1 3586.145,E2 3586.145} C_VEL
LIN {X 0,Y 544.271,Z 563.28,A -85,B 0,C 180,E1 3590.426,E2 3590.426} C_VEL
LIN {X 0,Y 544.36,Z 563.28,A -85,B 0,C 180,E1 3595.231,E2 3595.231} C_VEL
LIN {X 0,Y 544.43,Z 563.28,A -85,B 0,C 180,E1 3600.002,E2 3600.002} C_VEL
LIN {X 0,Y 544.416,Z 563.28,A -85,B 0,C 180,E1 3604.771,E2 3604.771} C_VEL
LIN {X 0,Y 544.332,Z 563.28,A -85,B 0,C 180,E1 3609.576,E2 3609.576} C_VEL
LIN {X 0,Y 544.311,Z 563.28,A -85,B 0,C 180,E1 3614.45,E2 3614.45} C_VEL
LIN {X 0,Y 544.222,Z 563.28,A -85,B 0,C 180,E1 3619.484,E2 3619.484} C_VEL
LIN {X 0,Y 544.083,Z 563.28,A -85,B 0,C 180,E1 3624.585,E2 3624.585} C_VEL
LIN {X 0,Y 544.06,Z 563.28,A -85,B 0,C 180,E1 3630.705,E2 3630.705} C_VEL
LIN {X 0,Y 544.125,Z 563.28,A -85,B 0,C 180,E1 3636.463,E2 3636.463} C_VEL
LIN {X 0,Y 544.031,Z 563.28,A -85,B 0,C 180,E1 3641.738,E2 3641.738} C_VEL
LIN {X 0,Y 544.027,Z 563.28,A -85,B 0,C 180,E1 3648.498,E2 3648.498} C_VEL
LIN {X 0,Y 544.15,Z 563.28,A -85,B 0,C 180,E1 3654.384,E2 3654.384} C_VEL
LIN {X 0,Y 544.117,Z 563.28,A -85,B 0,C 180,E1 3660.054,E2 3660.054} C_VEL
LIN {X 0,Y 544.053,Z 563.28,A -85,B 0,C 180,E1 3666.251,E2 3666.251} C_VEL
LIN {X 0,Y 544.243,Z 563.28,A -85,B 0,C 180,E1 3672.243,E2 3672.243} C_VEL
LIN {X 0,Y 544.324,Z 563.28,A -85,B 0,C 180,E1 3677.187,E2 3677.187} C_VEL
LIN {X 0,Y 544.387,Z 563.28,A -85,B 0,C 180,E1 3682.034,E2 3682.034} C_VEL
LIN {X 0,Y 544.513,Z 563.28,A -85,B 0,C 180,E1 3686.823,E2 3686.823} C_VEL
LIN {X 0,Y 544.631,Z 563.28,A -85,B 0,C 180,E1 3691.588,E2 3691.588} C_VEL
LIN {X 0,Y 544.533,Z 563.28,A -85,B 0,C 180,E1 3696.365,E2 3696.365} C_VEL
LIN {X 0,Y 544.323,Z 563.28,A -85,B 0,C 180,E1 3701.19,E2 3701.19} C_VEL
LIN {X 0,Y 544.236,Z 563.28,A -85,B 0,C 180,E1 3706.098,E2 3706.098} C_VEL
LIN {X 0,Y 544.183,Z 563.28,A -85,B 0,C 180,E1 3711.131,E2 3711.131} C_VEL
LIN {X 0,Y 544.022,Z 563.28,A -85,B 0,C 180,E1 3716.348,E2 3716.348} C_VEL
LIN {X 0,Y 543.977,Z 563.28,A -85,B 0,C 180,E1 3721.808,E2 3721.808} C_VEL
LIN {X 0,Y 544.176,Z 563.28,A -85,B 0,C 180,E1 3727.595,E2 3727.595} C_VEL
LIN {X 0,Y 543.962,Z 563.28,A -85,B 0,C 180,E1 3733.911,E2 3733.911} C_VEL
LIN {X 0,Y 544.051,Z 563.28,A -85,B 0,C 180,E1 3738.495,E2 3738.495} C_VEL
LIN {X 0,Y 543.973,Z 563.28,A -85,B 0,C 180,E1 3744.368,E2 3744.368} C_VEL
LIN {X 0,Y 543.98,Z 563.28,A -85,B 0,C 180,E1 3750.043,E2 3750.043} C_VEL
LIN {X 0,Y 544.118,Z 563.28,A -85,B 0,C 180,E1 3755.416,E2 3755.416} C_VEL
LIN {X 0,Y 544.292,Z 563.28,A -85,B 0,C 180,E1 3760.566,E2 3760.566} C_VEL
LIN {X 0,Y 543.996,Z 563.28,A -85,B 0,C 180,E1 3766.142,E2 3766.142} C_VEL
LIN {X 0,Y 544.27,Z 563.28,A -85,B 0,C 180,E1 3770.423,E2 3770.423} C_VEL
LIN {X 0,Y 544.377,Z 563.28,A -85,B 0,C 180,E1 3775.228,E2 3775.228} C_VEL
LIN {X 0,Y 544.45,Z 563.28,A -85,B 0,C 180,E1 3779.998,E2 3779.998} C_VEL
LIN {X 0,Y 544.426,Z 563.28,A -85,B 0,C 180,E1 3784.768,E2 3784.768} C_VEL
LIN {X 0,Y 544.349,Z 563.28,A -85,B 0,C 180,E1 3789.573,E2 3789.573} C_VEL
LIN {X 0,Y 544.343,Z 563.28,A -85,B 0,C 180,E1 3794.446,E2 3794.446} C_VEL
LIN {X 0,Y 544.183,Z 563.28,A -85,B 0,C 180,E1 3799.64,E2 3799.64} C_VEL
LIN {X 0,Y 544.082,Z 563.28,A -85,B 0,C 180,E1 3803.215,E2 3803.215} C_VEL
LIN {X 0,Y 540.129,Z 563.28,A -85,B 0,C 180,E1 3805.017,E2 3805.017} C_VEL
LIN {X 0,Y 536.089,Z 563.28,A -85,B 0,C 180,E1 3806.845,E2 3806.845} C_VEL
LIN {X 0,Y 536.233,Z 563.28,A -85,B 0,C 180,E1 3812.409,E2 3812.409} C_VEL
LIN {X 0,Y 536.154,Z 563.28,A -85,B 0,C 180,E1 3818.254,E2 3818.254} C_VEL
LIN {X 0,Y 535.892,Z 563.28,A -85,B 0,C 180,E1 3824.743,E2 3824.743} C_VEL
LIN {X 0,Y 536.04,Z 563.28,A -85,B 0,C 180,E1 3829.648,E2 3829.648} C_VEL
LIN {X 0,Y 536.273,Z 563.28,A -85,B 0,C 180,E1 3835.751,E2 3835.751} C_VEL
LIN {X 0,Y 536.35,Z 563.707,A -85,B 0,C 180,E1 3836.197,E2 3836.197} C_VEL
LIN {X 0,Y 547.189,Z 587.799,A -85,B 0,C 180,E1 3837.322,E2 3837.322} C_VEL
LIN {X 0,Y 546.638,Z 631.167,A -85,B 0,C 180,E1 3838.2,E2 3838.2} C_VEL
LIN {X 0,Y 545.269,Z 669.545,A -85,B 0,C 180,E1 3839.608,E2 3839.608} C_VEL
LIN {X 0,Y 543.555,Z 704.76,A -85,B 0,C 180,E1 3841.511,E2 3841.511} C_VEL
LIN {X 0,Y 541.565,Z 740.705,A -85,B 0,C 180,E1 3844.19,E2 3844.19} C_VEL
LIN {X 0,Y 539.79,Z 771.856,A -85,B 0,C 180,E1 3847.292,E2 3847.292} C_VEL
LIN {X 0,Y 538.384,Z 798.636,A -85,B 0,C 180,E1 3850.771,E2 3850.771} C_VEL
LIN {X 0,Y 537.424,Z 821.541,A -85,B 0,C 180,E1 3854.737,E2 3854.737} C_VEL
LIN {X 0,Y 536.953,Z 838.018,A -85,B 0,C 180,E1 3858.654,E2 3858.654} C_VEL
LIN {X 0,Y 536.813,Z 849.574,A -85,B 0,C 180,E1 3862.732,E2 3862.732} C_VEL
LIN {X 0,Y 536.754,Z 855.931,A -85,B 0,C 180,E1 3866.776,E2 3866.776} C_VEL
LIN {X 0,Y 536.694,Z 857.5,A -85,B 0,C 180,E1 3869.999,E2 3869.999} C_VEL
LIN {X 0,Y 536.647,Z 855.933,A -85,B 0,C 180,E1 3873.223,E2 3873.223} C_VEL
LIN {X 0,Y 536.792,Z 849.577,A -85,B 0,C 180,E1 3877.267,E2 3877.267} C_VEL
LIN {X 0,Y 536.95,Z 838.023,A -85,B 0,C 180,E1 3881.345,E2 3881.345} C_VEL
LIN {X 0,Y 537.555,Z 820.494,A -85,B 0,C 180,E1 3885.466,E2 3885.466} C_VEL
LIN {X 0,Y 538.531,Z 797.188,A -85,B 0,C 180,E1 3889.435,E2 3889.435} C_VEL
LIN {X 0,Y 540,Z 768.99,A -85,B 0,C 180,E1 3893.03,E2 3893.03} C_VEL
LIN {X 0,Y 541.723,Z 736.916,A -85,B 0,C 180,E1 3896.133,E2 3896.133} C_VEL
LIN {X 0,Y 543.702,Z 701.317,A -85,B 0,C 180,E1 3898.711,E2 3898.711} C_VEL
LIN {X 0,Y 545.562,Z 660.781,A -85,B 0,C 180,E1 3900.781,E2 3900.781} C_VEL
LIN {X 0,Y 546.875,Z 621.239,A -85,B 0,C 180,E1 3902.055,E2 3902.055} C_VEL
LIN {X 0,Y 546.768,Z 587.075,A -85,B 0,C 180,E1 3902.717,E2 3902.717} C_VEL
LIN {X 0,Y 536.099,Z 563.28,A -85,B 0,C 180,E1 3903.856,E2 3903.856} C_VEL
LIN {X 0,Y 536.171,Z 563.28,A -85,B 0,C 180,E1 3908.255,E2 3908.255} C_VEL
LIN {X 0,Y 535.962,Z 563.28,A -85,B 0,C 180,E1 3914.738,E2 3914.738} C_VEL
LIN {X 0,Y 536.054,Z 563.28,A -85,B 0,C 180,E1 3919.653,E2 3919.653} C_VEL
LIN {X 0,Y 535.994,Z 563.28,A -85,B 0,C 180,E1 3924.73,E2 3924.73} C_VEL
LIN {X 0,Y 536.013,Z 563.28,A -85,B 0,C 180,E1 3930.776,E2 3930.776} C_VEL
LIN {X 0,Y 536.174,Z 563.28,A -85,B 0,C 180,E1 3936.798,E2 3936.798} C_VEL
LIN {X 0,Y 536.376,Z 563.28,A -85,B 0,C 180,E1 3941.975,E2 3941.975} C_VEL
LIN {X 0,Y 536.322,Z 563.28,A -85,B 0,C 180,E1 3948.643,E2 3948.643} C_VEL
LIN {X 0,Y 536.577,Z 563.28,A -85,B 0,C 180,E1 3953.543,E2 3953.543} C_VEL
LIN {X 0,Y 536.714,Z 563.28,A -85,B 0,C 180,E1 3958.391,E2 3958.391} C_VEL
LIN {X 0,Y 536.502,Z 563.28,A -85,B 0,C 180,E1 3964.842,E2 3964.842} C_VEL
LIN {X 0,Y 536.362,Z 563.28,A -85,B 0,C 180,E1 3970.042,E2 3970.042} C_VEL
LIN {X 0,Y 536.373,Z 563.28,A -85,B 0,C 180,E1 3974.669,E2 3974.669} C_VEL
LIN {X 0,Y 536.311,Z 563.28,A -85,B 0,C 180,E1 3979.735,E2 3979.735} C_VEL
LIN {X 0,Y 536.086,Z 563.28,A -85,B 0,C 180,E1 3985.744,E2 3985.744} C_VEL
LIN {X 0,Y 536.145,Z 563.28,A -85,B 0,C 180,E1 3990.44,E2 3990.44} C_VEL
LIN {X 0,Y 536.22,Z 563.28,A -85,B 0,C 180,E1 3996.228,E2 3996.228} C_VEL
LIN {X 0,Y 536.015,Z 563.28,A -85,B 0,C 180,E1 4002.507,E2 4002.507} C_VEL
LIN {X 0,Y 536.008,Z 563.28,A -85,B 0,C 180,E1 4007.495,E2 4007.495} C_VEL
LIN {X 0,Y 536.225,Z 563.28,A -85,B 0,C 180,E1 4013.775,E2 4013.775} C_VEL
LIN {X 0,Y 536.24,Z 563.28,A -85,B 0,C 180,E1 4019.568,E2 4019.568} C_VEL
LIN {X 0,Y 536.094,Z 563.28,A -85,B 0,C 180,E1 4025.026,E2 4025.026} C_VEL
LIN {X 0,Y 536.257,Z 563.28,A -85,B 0,C 180,E1 4030.265,E2 4030.265} C_VEL
LIN {X 0,Y 536.377,Z 563.28,A -85,B 0,C 180,E1 4035.334,E2 4035.334} C_VEL
LIN {X 0,Y 536.436,Z 563.28,A -85,B 0,C 180,E1 4040.284,E2 4040.284} C_VEL
LIN {X 0,Y 536.619,Z 563.28,A -85,B 0,C 180,E1 4046.777,E2 4046.777} C_VEL
LIN {X 0,Y 536.73,Z 563.28,A -85,B 0,C 180,E1 4051.612,E2 4051.612} C_VEL
LIN {X 0,Y 536.602,Z 563.28,A -85,B 0,C 180,E1 4056.459,E2 4056.459} C_VEL
LIN {X 0,Y 536.41,Z 563.28,A -85,B 0,C 180,E1 4061.358,E2 4061.358} C_VEL
LIN {X 0,Y 536.264,Z 563.28,A -85,B 0,C 180,E1 4066.912,E2 4066.912} C_VEL
LIN {X 0,Y 536.218,Z 563.28,A -85,B 0,C 180,E1 4071.768,E2 4071.768} C_VEL
LIN {X 0,Y 536.079,Z 563.28,A -85,B 0,C 180,E1 4076.769,E2 4076.769} C_VEL
LIN {X 0,Y 536.041,Z 563.28,A -85,B 0,C 180,E1 4082.377,E2 4082.377} C_VEL
LIN {X 0,Y 536.207,Z 563.28,A -85,B 0,C 180,E1 4088.254,E2 4088.254} C_VEL
LIN {X 0,Y 535.994,Z 563.28,A -85,B 0,C 180,E1 4094.737,E2 4094.737} C_VEL
LIN {X 0,Y 536.067,Z 563.28,A -85,B 0,C 180,E1 4099.65,E2 4099.65} C_VEL
LIN {X 0,Y 536.02,Z 563.28,A -85,B 0,C 180,E1 4104.729,E2 4104.729} C_VEL
LIN {X 0,Y 536.033,Z 563.28,A -85,B 0,C 180,E1 4110.775,E2 4110.775} C_VEL
LIN {X 0,Y 536.203,Z 563.28,A -85,B 0,C 180,E1 4116.795,E2 4116.795} C_VEL
LIN {X 0,Y 536.378,Z 563.28,A -85,B 0,C 180,E1 4121.971,E2 4121.971} C_VEL
LIN {X 0,Y 536.311,Z 563.28,A -85,B 0,C 180,E1 4128.639,E2 4128.639} C_VEL
LIN {X 0,Y 536.594,Z 563.28,A -85,B 0,C 180,E1 4133.54,E2 4133.54} C_VEL
LIN {X 0,Y 536.739,Z 563.28,A -85,B 0,C 180,E1 4138.387,E2 4138.387} C_VEL
LIN {X 0,Y 536.512,Z 563.28,A -85,B 0,C 180,E1 4144.839,E2 4144.839} C_VEL
LIN {X 0,Y 536.407,Z 563.28,A -85,B 0,C 180,E1 4150.06,E2 4150.06} C_VEL
LIN {X 0,Y 536.396,Z 563.28,A -85,B 0,C 180,E1 4154.664,E2 4154.664} C_VEL
LIN {X 0,Y 536.296,Z 563.28,A -85,B 0,C 180,E1 4159.732,E2 4159.732} C_VEL
LIN {X 0,Y 536.073,Z 563.28,A -85,B 0,C 180,E1 4165.738,E2 4165.738} C_VEL
LIN {X 0,Y 536.089,Z 563.28,A -85,B 0,C 180,E1 4166.845,E2 4166.845} C_VEL
LIN {X 0,Y 532.037,Z 563.28,A -85,B 0,C 180,E1 4168.676,E2 4168.676} C_VEL
LIN {X 0,Y 528.163,Z 563.28,A -85,B 0,C 180,E1 4170.534,E2 4170.534} C_VEL
LIN {X 0,Y 528.328,Z 563.28,A -85,B 0,C 180,E1 4174.834,E2 4174.834} C_VEL
LIN {X 0,Y 528.037,Z 563.28,A -85,B 0,C 180,E1 4181.09,E2 4181.09} C_VEL
LIN {X 0,Y 528.013,Z 563.28,A -85,B 0,C 180,E1 4186.693,E2 4186.693} C_VEL
LIN {X 0,Y 528.241,Z 563.28,A -85,B 0,C 180,E1 4193.136,E2 4193.136} C_VEL
LIN {X 0,Y 528.355,Z 563.28,A -85,B 0,C 180,E1 4195.607,E2 4195.607} C_VEL
LIN {X 0,Y 540.706,Z 592.019,A -85,B 0,C 180,E1 4196.946,E2 4196.946} C_VEL
LIN {X 0,Y 539.849,Z 632.479,A -85,B 0,C 180,E1 4197.796,E2 4197.796} C_VEL
LIN {X 0,Y 538.274,Z 672.067,A -85,B 0,C 180,E1 4199.292,E2 4199.292} C_VEL
LIN {X 0,Y 536.259,Z 708.433,A -85,B 0,C 180,E1 4201.343,E2 4201.343} C_VEL
LIN {X 0,Y 534.131,Z 743.214,A -85,B 0,C 180,E1 4204.03,E2 4204.03} C_VEL
LIN {X 0,Y 532.069,Z 775.912,A -85,B 0,C 180,E1 4207.426,E2 4207.426} C_VEL
LIN {X 0,Y 530.569,Z 802.66,A -85,B 0,C 180,E1 4211.123,E2 4211.123} C_VEL
LIN {X 0,Y 529.6,Z 824.525,A -85,B 0,C 180,E1 4215.14,E2 4215.14} C_VEL
LIN {X 0,Y 529.122,Z 841.022,A -85,B 0,C 180,E1 4219.403,E2 4219.403} C_VEL
LIN {X 0,Y 528.92,Z 851.242,A -85,B 0,C 180,E1 4223.446,E2 4223.446} C_VEL
LIN {X 0,Y 528.838,Z 856.207,A -85,B 0,C 180,E1 4227.033,E2 4227.033} C_VEL
LIN {X 0,Y 528.892,Z 857.106,A -85,B 0,C 180,E1 4231.634,E2 4231.634} C_VEL
LIN {X 0,Y 528.872,Z 852.723,A -85,B 0,C 180,E1 4235.731,E2 4235.731} C_VEL
LIN {X 0,Y 528.962,Z 843.29,A -85,B 0,C 180,E1 4239.855,E2 4239.855} C_VEL
LIN {X 0,Y 529.385,Z 829.478,A -85,B 0,C 180,E1 4243.741,E2 4243.741} C_VEL
LIN {X 0,Y 530.142,Z 810.272,A -85,B 0,C 180,E1 4247.616,E2 4247.616} C_VEL
LIN {X 0,Y 531.466,Z 786.098,A -85,B 0,C 180,E1 4251.286,E2 4251.286} C_VEL
LIN {X 0,Y 533.372,Z 755.292,A -85,B 0,C 180,E1 4254.829,E2 4254.829} C_VEL
LIN {X 0,Y 535.479,Z 720.968,A -85,B 0,C 180,E1 4257.781,E2 4257.781} C_VEL
LIN {X 0,Y 537.589,Z 685.268,A -85,B 0,C 180,E1 4260.043,E2 4260.043} C_VEL
LIN {X 0,Y 539.396,Z 646.989,A -85,B 0,C 180,E1 4261.735,E2 4261.735} C_VEL
LIN {X 0,Y 540.561,Z 610.772,A -85,B 0,C 180,E1 4262.729,E2 4262.729} C_VEL
LIN {X 0,Y 539.959,Z 589.172,A -85,B 0,C 180,E1 4263.15,E2 4263.15} C_VEL
LIN {X 0,Y 528.177,Z 563.28,A -85,B 0,C 180,E1 4264.487,E2 4264.487} C_VEL
LIN {X 0,Y 528.103,Z 563.28,A -85,B 0,C 180,E1 4269.515,E2 4269.515} C_VEL
LIN {X 0,Y 528.08,Z 563.28,A -85,B 0,C 180,E1 4275.592,E2 4275.592} C_VEL
LIN {X 0,Y 528.121,Z 563.28,A -85,B 0,C 180,E1 4281.055,E2 4281.055} C_VEL
LIN {X 0,Y 528.064,Z 563.28,A -85,B 0,C 180,E1 4287.118,E2 4287.118} C_VEL
LIN {X 0,Y 528.158,Z 563.28,A -85,B 0,C 180,E1 4292.8,E2 4292.8} C_VEL
LIN {X 0,Y 528.319,Z 563.28,A -85,B 0,C 180,E1 4298.206,E2 4298.206} C_VEL
LIN {X 0,Y 528.411,Z 563.28,A -85,B 0,C 180,E1 4303.409,E2 4303.409} C_VEL
LIN {X 0,Y 528.461,Z 563.28,A -85,B 0,C 180,E1 4310.137,E2 4310.137} C_VEL
LIN {X 0,Y 528.576,Z 563.28,A -85,B 0,C 180,E1 4315.089,E2 4315.089} C_VEL
LIN {X 0,Y 528.636,Z 563.28,A -85,B 0,C 180,E1 4320.002,E2 4320.002} C_VEL
LIN {X 0,Y 528.604,Z 563.28,A -85,B 0,C 180,E1 4324.915,E2 4324.915} C_VEL
LIN {X 0,Y 528.494,Z 563.28,A -85,B 0,C 180,E1 4329.866,E2 4329.866} C_VEL
LIN {X 0,Y 528.463,Z 563.28,A -85,B 0,C 180,E1 4334.893,E2 4334.893} C_VEL
LIN {X 0,Y 528.379,Z 563.28,A -85,B 0,C 180,E1 4340.044,E2 4340.044} C_VEL
LIN {X 0,Y 528.209,Z 563.28,A -85,B 0,C 180,E1 4345.376,E2 4345.376} C_VEL
LIN {X 0,Y 528.219,Z 563.28,A -85,B 0,C 180,E1 4351.016,E2 4351.016} C_VEL
LIN {X 0,Y 528.255,Z 563.28,A -85,B 0,C 180,E1 4356.863,E2 4356.863} C_VEL
LIN {X 0,Y 528.042,Z 563.28,A -85,B 0,C 180,E1 4363.305,E2 4363.305} C_VEL
LIN {X 0,Y 528.077,Z 563.28,A -85,B 0,C 180,E1 4368.912,E2 4368.912} C_VEL
LIN {X 0,Y 528.321,Z 563.28,A -85,B 0,C 180,E1 4375.164,E2 4375.164} C_VEL
LIN {X 0,Y 528.267,Z 563.28,A -85,B 0,C 180,E1 4380.948,E2 4380.948} C_VEL
LIN {X 0,Y 528.185,Z 563.28,A -85,B 0,C 180,E1 4386.424,E2 4386.424} C_VEL
LIN {X 0,Y 528.369,Z 563.28,A -85,B 0,C 180,E1 4391.691,E2 4391.691} C_VEL
LIN {X 0,Y 528.509,Z 563.28,A -85,B 0,C 180,E1 4396.797,E2 4396.797} C_VEL
LIN {X 0,Y 528.562,Z 563.28,A -85,B 0,C 180,E1 4401.794,E2 4401.794} C_VEL
LIN {X 0,Y 528.539,Z 563.28,A -85,B 0,C 180,E1 4407.831,E2 4407.831} C_VEL
LIN {X 0,Y 528.583,Z 563.28,A -85,B 0,C 180,E1 4413.274,E2 4413.274} C_VEL
LIN {X 0,Y 528.455,Z 563.28,A -85,B 0,C 180,E1 4418.209,E2 4418.209} C_VEL
LIN {X 0,Y 528.355,Z 563.28,A -85,B 0,C 180,E1 4423.815,E2 4423.815} C_VEL
LIN {X 0,Y 528.38,Z 563.28,A -85,B 0,C 180,E1 4429.53,E2 4429.53} C_VEL
LIN {X 0,Y 528.215,Z 563.28,A -85,B 0,C 180,E1 4435.375,E2 4435.375} C_VEL
LIN {X 0,Y 528.095,Z 563.28,A -85,B 0,C 180,E1 4440.99,E2 4440.99} C_VEL
LIN {X 0,Y 528.237,Z 563.28,A -85,B 0,C 180,E1 4446.88,E2 4446.88} C_VEL
LIN {X 0,Y 528.035,Z 563.28,A -85,B 0,C 180,E1 4453.305,E2 4453.305} C_VEL
LIN {X 0,Y 528.1,Z 563.28,A -85,B 0,C 180,E1 4458.911,E2 4458.911} C_VEL
LIN {X 0,Y 528.085,Z 563.28,A -85,B 0,C 180,E1 4465.144,E2 4465.144} C_VEL
LIN {X 0,Y 528.163,Z 563.28,A -85,B 0,C 180,E1 4470.94,E2 4470.94} C_VEL
LIN {X 0,Y 528.254,Z 563.28,A -85,B 0,C 180,E1 4476.425,E2 4476.425} C_VEL
LIN {X 0,Y 528.443,Z 563.28,A -85,B 0,C 180,E1 4481.691,E2 4481.691} C_VEL
LIN {X 0,Y 528.366,Z 563.28,A -85,B 0,C 180,E1 4488.466,E2 4488.466} C_VEL
LIN {X 0,Y 528.672,Z 563.28,A -85,B 0,C 180,E1 4493.442,E2 4493.442} C_VEL
LIN {X 0,Y 528.829,Z 563.28,A -85,B 0,C 180,E1 4498.363,E2 4498.363} C_VEL
LIN {X 0,Y 528.613,Z 563.28,A -85,B 0,C 180,E1 4504.911,E2 4504.911} C_VEL
LIN {X 0,Y 528.525,Z 563.28,A -85,B 0,C 180,E1 4509.862,E2 4509.862} C_VEL
LIN {X 0,Y 528.476,Z 563.28,A -85,B 0,C 180,E1 4514.889,E2 4514.889} C_VEL
LIN {X 0,Y 528.365,Z 563.28,A -85,B 0,C 180,E1 4520.04,E2 4520.04} C_VEL
LIN {X 0,Y 528.197,Z 563.28,A -85,B 0,C 180,E1 4525.372,E2 4525.372} C_VEL
LIN {X 0,Y 528.163,Z 563.28,A -85,B 0,C 180,E1 4530.534,E2 4530.534} C_VEL
LIN {X 0,Y 525.724,Z 563.28,A -85,B 0,C 180,E1 4531.937,E2 4531.937} C_VEL
LIN {X 0,Y 520.296,Z 563.28,A -85,B 0,C 180,E1 4534.284,E2 4534.284} C_VEL
LIN {X 0,Y 520.198,Z 563.28,A -85,B 0,C 180,E1 4539.653,E2 4539.653} C_VEL
LIN {X 0,Y 520.081,Z 563.28,A -85,B 0,C 180,E1 4545.863,E2 4545.863} C_VEL
LIN {X 0,Y 520.221,Z 563.28,A -85,B 0,C 180,E1 4551.55,E2 4551.55} C_VEL
LIN {X 0,Y 520.434,Z 563.561,A -85,B 0,C 180,E1 4555.013,E2 4555.013} C_VEL
LIN {X 0,Y 534.069,Z 592.976,A -85,B 0,C 180,E1 4556.496,E2 4556.496} C_VEL
LIN {X 0,Y 533.156,Z 632.456,A -85,B 0,C 180,E1 4557.342,E2 4557.342} C_VEL
LIN {X 0,Y 531.463,Z 671.358,A -85,B 0,C 180,E1 4558.819,E2 4558.819} C_VEL
LIN {X 0,Y 529.255,Z 707.333,A -85,B 0,C 180,E1 4560.85,E2 4560.85} C_VEL
LIN {X 0,Y 526.937,Z 741.962,A -85,B 0,C 180,E1 4563.533,E2 4563.533} C_VEL
LIN {X 0,Y 524.664,Z 773.914,A -85,B 0,C 180,E1 4566.849,E2 4566.849} C_VEL
LIN {X 0,Y 522.948,Z 799.981,A -85,B 0,C 180,E1 4570.399,E2 4570.399} C_VEL
LIN {X 0,Y 521.783,Z 822.569,A -85,B 0,C 180,E1 4574.483,E2 4574.483} C_VEL
LIN {X 0,Y 521.209,Z 838.012,A -85,B 0,C 180,E1 4578.306,E2 4578.306} C_VEL
LIN {X 0,Y 521.009,Z 849.568,A -85,B 0,C 180,E1 4582.51,E2 4582.51} C_VEL
LIN {X 0,Y 520.954,Z 855.937,A -85,B 0,C 180,E1 4586.678,E2 4586.678} C_VEL
LIN {X 0,Y 520.901,Z 857.5,A -85,B 0,C 180,E1 4589.999,E2 4589.999} C_VEL
LIN {X 0,Y 520.868,Z 855.939,A -85,B 0,C 180,E1 4593.321,E2 4593.321} C_VEL
LIN {X 0,Y 521.007,Z 849.571,A -85,B 0,C 180,E1 4597.488,E2 4597.488} C_VEL
LIN {X 0,Y 521.252,Z 838.017,A -85,B 0,C 180,E1 4601.691,E2 4601.691} C_VEL
LIN {X 0,Y 521.997,Z 820.484,A -85,B 0,C 180,E1 4605.939,E2 4605.939} C_VEL
LIN {X 0,Y 523.201,Z 797.192,A -85,B 0,C 180,E1 4610.028,E2 4610.028} C_VEL
LIN {X 0,Y 525.062,Z 768.996,A -85,B 0,C 180,E1 4613.725,E2 4613.725} C_VEL
LIN {X 0,Y 527.22,Z 736.899,A -85,B 0,C 180,E1 4616.909,E2 4616.909} C_VEL
LIN {X 0,Y 529.66,Z 701.496,A -85,B 0,C 180,E1 4619.534,E2 4619.534} C_VEL
LIN {X 0,Y 531.906,Z 661.397,A -85,B 0,C 180,E1 4621.63,E2 4621.63} C_VEL
LIN {X 0,Y 533.459,Z 622.809,A -85,B 0,C 180,E1 4622.919,E2 4622.919} C_VEL
LIN {X 0,Y 533.429,Z 592.028,A -85,B 0,C 180,E1 4623.564,E2 4623.564} C_VEL
LIN {X 0,Y 520.231,Z 563.28,A -85,B 0,C 180,E1 4625.046,E2 4625.046} C_VEL
LIN {X 0,Y 520.135,Z 563.28,A -85,B 0,C 180,E1 4631.039,E2 4631.039} C_VEL
LIN {X 0,Y 520.164,Z 563.28,A -85,B 0,C 180,E1 4636.489,E2 4636.489} C_VEL
LIN {X 0,Y 520.156,Z 563.28,A -85,B 0,C 180,E1 4642.469,E2 4642.469} C_VEL
LIN {X 0,Y 520.156,Z 563.28,A -85,B 0,C 180,E1 4648.523,E2 4648.523} C_VEL
LIN {X 0,Y 520.271,Z 563.28,A -85,B 0,C 180,E1 4654.213,E2 4654.213} C_VEL
LIN {X 0,Y 520.442,Z 563.28,A -85,B 0,C 180,E1 4659.641,E2 4659.641} C_VEL
LIN {X 0,Y 520.323,Z 563.28,A -85,B 0,C 180,E1 4664.872,E2 4664.872} C_VEL
LIN {X 0,Y 520.542,Z 563.28,A -85,B 0,C 180,E1 4670.271,E2 4670.271} C_VEL
LIN {X 0,Y 520.671,Z 563.28,A -85,B 0,C 180,E1 4675.014,E2 4675.014} C_VEL
LIN {X 0,Y 520.748,Z 563.28,A -85,B 0,C 180,E1 4680.002,E2 4680.002} C_VEL
LIN {X 0,Y 520.69,Z 563.28,A -85,B 0,C 180,E1 4684.989,E2 4684.989} C_VEL
LIN {X 0,Y 520.588,Z 563.28,A -85,B 0,C 180,E1 4690.017,E2 4690.017} C_VEL
LIN {X 0,Y 520.531,Z 563.28,A -85,B 0,C 180,E1 4695.126,E2 4695.126} C_VEL
LIN {X 0,Y 520.435,Z 563.28,A -85,B 0,C 180,E1 4700.363,E2 4700.363} C_VEL
LIN {X 0,Y 520.248,Z 563.28,A -85,B 0,C 180,E1 4705.952,E2 4705.952} C_VEL
LIN {X 0,Y 520.307,Z 563.28,A -85,B 0,C 180,E1 4711.471,E2 4711.471} C_VEL
LIN {X 0,Y 520.276,Z 563.28,A -85,B 0,C 180,E1 4717.525,E2 4717.525} C_VEL
LIN {X 0,Y 520.127,Z 563.28,A -85,B 0,C 180,E1 4723.507,E2 4723.507} C_VEL
LIN {X 0,Y 520.173,Z 563.28,A -85,B 0,C 180,E1 4728.962,E2 4728.962} C_VEL
LIN {X 0,Y 520.332,Z 563.28,A -85,B 0,C 180,E1 4734.549,E2 4734.549} C_VEL
LIN {X 0,Y 520.339,Z 563.28,A -85,B 0,C 180,E1 4740.462,E2 4740.462} C_VEL
LIN {X 0,Y 520.279,Z 563.28,A -85,B 0,C 180,E1 4746.044,E2 4746.044} C_VEL
LIN {X 0,Y 520.456,Z 563.28,A -85,B 0,C 180,E1 4751.402,E2 4751.402} C_VEL
LIN {X 0,Y 520.616,Z 563.28,A -85,B 0,C 180,E1 4756.593,E2 4756.593} C_VEL
LIN {X 0,Y 520.643,Z 563.28,A -85,B 0,C 180,E1 4761.668,E2 4761.668} C_VEL
LIN {X 0,Y 520.828,Z 563.28,A -85,B 0,C 180,E1 4766.679,E2 4766.679} C_VEL
LIN {X 0,Y 520.926,Z 563.28,A -85,B 0,C 180,E1 4771.661,E2 4771.661} C_VEL
LIN {X 0,Y 520.751,Z 563.28,A -85,B 0,C 180,E1 4776.657,E2 4776.657} C_VEL
LIN {X 0,Y 520.559,Z 563.28,A -85,B 0,C 180,E1 4781.708,E2 4781.708} C_VEL
LIN {X 0,Y 520.455,Z 563.28,A -85,B 0,C 180,E1 4786.899,E2 4786.899} C_VEL
LIN {X 0,Y 520.392,Z 563.28,A -85,B 0,C 180,E1 4792.147,E2 4792.147} C_VEL
LIN {X 0,Y 520.221,Z 563.28,A -85,B 0,C 180,E1 4797.654,E2 4797.654} C_VEL
LIN {X 0,Y 520.187,Z 563.28,A -85,B 0,C 180,E1 4803.448,E2 4803.448} C_VEL
LIN {X 0,Y 520.237,Z 563.28,A -85,B 0,C 180,E1 4809.654,E2 4809.654} C_VEL
LIN {X 0,Y 520.187,Z 563.28,A -85,B 0,C 180,E1 4815.874,E2 4815.874} C_VEL
LIN {X 0,Y 520.207,Z 563.28,A -85,B 0,C 180,E1 4821.557,E2 4821.557} C_VEL
LIN {X 0,Y 520.161,Z 563.28,A -85,B 0,C 180,E1 4827.279,E2 4827.279} C_VEL
LIN {X 0,Y 520.271,Z 563.28,A -85,B 0,C 180,E1 4832.349,E2 4832.349} C_VEL
LIN {X 0,Y 520.428,Z 563.28,A -85,B 0,C 180,E1 4838.105,E2 4838.105} C_VEL
LIN {X 0,Y 520.52,Z 563.28,A -85,B 0,C 180,E1 4843.146,E2 4843.146} C_VEL
LIN {X 0,Y 520.541,Z 563.28,A -85,B 0,C 180,E1 4850.281,E2 4850.281} C_VEL
LIN {X 0,Y 520.688,Z 563.28,A -85,B 0,C 180,E1 4855.011,E2 4855.011} C_VEL
LIN {X 0,Y 520.766,Z 563.28,A -85,B 0,C 180,E1 4859.998,E2 4859.998} C_VEL
LIN {X 0,Y 520.699,Z 563.28,A -85,B 0,C 180,E1 4864.986,E2 4864.986} C_VEL
LIN {X 0,Y 520.627,Z 563.28,A -85,B 0,C 180,E1 4870.013,E2 4870.013} C_VEL
LIN {X 0,Y 520.535,Z 563.28,A -85,B 0,C 180,E1 4875.122,E2 4875.122} C_VEL
LIN {X 0,Y 520.421,Z 563.28,A -85,B 0,C 180,E1 4880.36,E2 4880.36} C_VEL
LIN {X 0,Y 520.236,Z 563.28,A -85,B 0,C 180,E1 4885.946,E2 4885.946} C_VEL
LIN {X 0,Y 520.31,Z 563.28,A -85,B 0,C 180,E1 4891.466,E2 4891.466} C_VEL
LIN {X 0,Y 520.296,Z 563.28,A -85,B 0,C 180,E1 4894.284,E2 4894.284} C_VEL
LIN {X 0,Y 519.001,Z 563.28,A -85,B 0,C 180,E1 4895.237,E2 4895.237} C_VEL
LIN {X 0,Y 512.406,Z 563.28,A -85,B 0,C 180,E1 4897.832,E2 4897.832} C_VEL
LIN {X 0,Y 512.319,Z 563.28,A -85,B 0,C 180,E1 4898.078,E2 4898.078} C_VEL
LIN {X 0,Y 512.153,Z 563.28,A -85,B 0,C 180,E1 4902.659,E2 4902.659} C_VEL
LIN {X 0,Y 512.256,Z 563.28,A -85,B 0,C 180,E1 4909.602,E2 4909.602} C_VEL
LIN {X 0,Y 512.457,Z 563.28,A -85,B 0,C 180,E1 4914.361,E2 4914.361} C_VEL
LIN {X 0,Y 527.463,Z 595.398,A -85,B 0,C 180,E1 4916.059,E2 4916.059} C_VEL
LIN {X 0,Y 526.319,Z 636.199,A -85,B 0,C 180,E1 4916.992,E2 4916.992} C_VEL
LIN {X 0,Y 524.42,Z 674.881,A -85,B 0,C 180,E1 4918.534,E2 4918.534} C_VEL
LIN {X 0,Y 521.962,Z 711.135,A -85,B 0,C 180,E1 4920.68,E2 4920.68} C_VEL
LIN {X 0,Y 519.517,Z 744.372,A -85,B 0,C 180,E1 4923.358,E2 4923.358} C_VEL
LIN {X 0,Y 517.027,Z 776.506,A -85,B 0,C 180,E1 4926.806,E2 4926.806} C_VEL
LIN {X 0,Y 515.117,Z 802.713,A -85,B 0,C 180,E1 4930.544,E2 4930.544} C_VEL
LIN {X 0,Y 513.958,Z 822.571,A -85,B 0,C 180,E1 4934.241,E2 4934.241} C_VEL
LIN {X 0,Y 513.34,Z 838.009,A -85,B 0,C 180,E1 4938.125,E2 4938.125} C_VEL
LIN {X 0,Y 513.108,Z 849.565,A -85,B 0,C 180,E1 4942.394,E2 4942.394} C_VEL
LIN {X 0,Y 513.076,Z 855.94,A -85,B 0,C 180,E1 4946.627,E2 4946.627} C_VEL
LIN {X 0,Y 513.003,Z 857.5,A -85,B 0,C 180,E1 4949.999,E2 4949.999} C_VEL
LIN {X 0,Y 512.983,Z 855.941,A -85,B 0,C 180,E1 4953.372,E2 4953.372} C_VEL
LIN {X 0,Y 513.114,Z 849.569,A -85,B 0,C 180,E1 4957.604,E2 4957.604} C_VEL
LIN {X 0,Y 513.407,Z 838.014,A -85,B 0,C 180,E1 4961.872,E2 4961.872} C_VEL
LIN {X 0,Y 514.225,Z 820.48,A -85,B 0,C 180,E1 4966.187,E2 4966.187} C_VEL
LIN {X 0,Y 515.462,Z 798.694,A -85,B 0,C 180,E1 4970.111,E2 4970.111} C_VEL
LIN {X 0,Y 517.466,Z 770.868,A -85,B 0,C 180,E1 4973.865,E2 4973.865} C_VEL
LIN {X 0,Y 519.795,Z 739.468,A -85,B 0,C 180,E1 4977.091,E2 4977.091} C_VEL
LIN {X 0,Y 522.549,Z 703.259,A -85,B 0,C 180,E1 4979.855,E2 4979.855} C_VEL
LIN {X 0,Y 524.902,Z 664.299,A -85,B 0,C 180,E1 4981.96,E2 4981.96} C_VEL
LIN {X 0,Y 526.705,Z 626.309,A -85,B 0,C 180,E1 4983.302,E2 4983.302} C_VEL
LIN {X 0,Y 527.096,Z 595.042,A -85,B 0,C 180,E1 4983.974,E2 4983.974} C_VEL
LIN {X 0,Y 512.331,Z 563.28,A -85,B 0,C 180,E1 4985.657,E2 4985.657} C_VEL
LIN {X 0,Y 512.246,Z 563.28,A -85,B 0,C 180,E1 4990.397,E2 4990.397} C_VEL
LIN {X 0,Y 512.204,Z 563.28,A -85,B 0,C 180,E1 4995.007,E2 4995.007} C_VEL
LIN {X 0,Y 512.283,Z 563.28,A -85,B 0,C 180,E1 4999.983,E2 4999.983} C_VEL
LIN {X 0,Y 512.165,Z 563.28,A -85,B 0,C 180,E1 5005.961,E2 5005.961} C_VEL
LIN {X 0,Y 512.31,Z 563.28,A -85,B 0,C 180,E1 5012.084,E2 5012.084} C_VEL
LIN {X 0,Y 512.426,Z 563.28,A -85,B 0,C 180,E1 5017.493,E2 5017.493} C_VEL
LIN {X 0,Y 512.588,Z 563.28,A -85,B 0,C 180,E1 5022.881,E2 5022.881} C_VEL
LIN {X 0,Y 512.616,Z 563.28,A -85,B 0,C 180,E1 5029.829,E2 5029.829} C_VEL
LIN {X 0,Y 512.79,Z 563.28,A -85,B 0,C 180,E1 5034.937,E2 5034.937} C_VEL
LIN {X 0,Y 512.852,Z 563.28,A -85,B 0,C 180,E1 5040.002,E2 5040.002} C_VEL
LIN {X 0,Y 512.8,Z 563.28,A -85,B 0,C 180,E1 5045.066,E2 5045.066} C_VEL
LIN {X 0,Y 512.664,Z 563.28,A -85,B 0,C 180,E1 5050.174,E2 5050.174} C_VEL
LIN {X 0,Y 512.6,Z 563.28,A -85,B 0,C 180,E1 5055.365,E2 5055.365} C_VEL
LIN {X 0,Y 512.531,Z 563.28,A -85,B 0,C 180,E1 5060.691,E2 5060.691} C_VEL
LIN {X 0,Y 512.334,Z 563.28,A -85,B 0,C 180,E1 5066.221,E2 5066.221} C_VEL
LIN {X 0,Y 512.44,Z 563.28,A -85,B 0,C 180,E1 5072.011,E2 5072.011} C_VEL
LIN {X 0,Y 512.338,Z 563.28,A -85,B 0,C 180,E1 5078.21,E2 5078.21} C_VEL
LIN {X 0,Y 512.177,Z 563.28,A -85,B 0,C 180,E1 5085.001,E2 5085.001} C_VEL
LIN {X 0,Y 512.337,Z 563.28,A -85,B 0,C 180,E1 5091.793,E2 5091.793} C_VEL
LIN {X 0,Y 512.478,Z 563.28,A -85,B 0,C 180,E1 5097.994,E2 5097.994} C_VEL
LIN {X 0,Y 512.31,Z 563.28,A -85,B 0,C 180,E1 5103.781,E2 5103.781} C_VEL
LIN {X 0,Y 512.455,Z 563.28,A -85,B 0,C 180,E1 5109.308,E2 5109.308} C_VEL
LIN {X 0,Y 512.596,Z 563.28,A -85,B 0,C 180,E1 5114.637,E2 5114.637} C_VEL
LIN {X 0,Y 512.702,Z 563.28,A -85,B 0,C 180,E1 5119.829,E2 5119.829} C_VEL
LIN {X 0,Y 512.815,Z 563.28,A -85,B 0,C 180,E1 5124.936,E2 5124.936} C_VEL
LIN {X 0,Y 513.029,Z 563.28,A -85,B 0,C 180,E1 5131.686,E2 5131.686} C_VEL
LIN {X 0,Y 512.823,Z 563.28,A -85,B 0,C 180,E1 5136.76,E2 5136.76} C_VEL
LIN {X 0,Y 512.631,Z 563.28,A -85,B 0,C 180,E1 5141.892,E2 5141.892} C_VEL
LIN {X 0,Y 512.552,Z 563.28,A -85,B 0,C 180,E1 5147.123,E2 5147.123} C_VEL
LIN {X 0,Y 512.438,Z 563.28,A -85,B 0,C 180,E1 5152.509,E2 5152.509} C_VEL
LIN {X 0,Y 512.273,Z 563.28,A -85,B 0,C 180,E1 5158.121,E2 5158.121} C_VEL
LIN {X 0,Y 512.231,Z 563.28,A -85,B 0,C 180,E1 5164.423,E2 5164.423} C_VEL
LIN {X 0,Y 512.277,Z 563.28,A -85,B 0,C 180,E1 5170.396,E2 5170.396} C_VEL
LIN {X 0,Y 512.237,Z 563.28,A -85,B 0,C 180,E1 5175.005,E2 5175.005} C_VEL
LIN {X 0,Y 512.301,Z 563.28,A -85,B 0,C 180,E1 5179.983,E2 5179.983} C_VEL
LIN {X 0,Y 512.185,Z 563.28,A -85,B 0,C 180,E1 5185.958,E2 5185.958} C_VEL
LIN {X 0,Y 512.329,Z 563.28,A -85,B 0,C 180,E1 5192.084,E2 5192.084} C_VEL
LIN {X 0,Y 512.452,Z 563.28,A -85,B 0,C 180,E1 5197.491,E2 5197.491} C_VEL
LIN {X 0,Y 512.61,Z 563.28,A -85,B 0,C 180,E1 5202.878,E2 5202.878} C_VEL
LIN {X 0,Y 512.613,Z 563.28,A -85,B 0,C 180,E1 5209.825,E2 5209.825} C_VEL
LIN {X 0,Y 512.807,Z 563.28,A -85,B 0,C 180,E1 5214.934,E2 5214.934} C_VEL
LIN {X 0,Y 512.868,Z 563.28,A -85,B 0,C 180,E1 5219.998,E2 5219.998} C_VEL
LIN {X 0,Y 512.809,Z 563.28,A -85,B 0,C 180,E1 5225.063,E2 5225.063} C_VEL
LIN {X 0,Y 512.702,Z 563.28,A -85,B 0,C 180,E1 5230.17,E2 5230.17} C_VEL
LIN {X 0,Y 512.595,Z 563.28,A -85,B 0,C 180,E1 5235.362,E2 5235.362} C_VEL
LIN {X 0,Y 512.522,Z 563.28,A -85,B 0,C 180,E1 5240.688,E2 5240.688} C_VEL
LIN {X 0,Y 512.321,Z 563.28,A -85,B 0,C 180,E1 5246.217,E2 5246.217} C_VEL
LIN {X 0,Y 512.445,Z 563.28,A -85,B 0,C 180,E1 5252.006,E2 5252.006} C_VEL
LIN {X 0,Y 512.319,Z 563.28,A -85,B 0,C 180,E1 5258.078,E2 5258.078} C_VEL
LIN {X 0,Y 509.783,Z 563.28,A -85,B 0,C 180,E1 5259.507,E2 5259.507} C_VEL
LIN {X 0,Y 504.156,Z 563.28,A -85,B 0,C 180,E1 5261.894,E2 5261.894} C_VEL
LIN {X 0,Y 504.223,Z 563.28,A -85,B 0,C 180,E1 5268.43,E2 5268.43} C_VEL
LIN {X 0,Y 504.481,Z 563.28,A -85,B 0,C 180,E1 5273.727,E2 5273.727} C_VEL
LIN {X 0,Y 515.234,Z 586.019,A -85,B 0,C 180,E1 5274.984,E2 5274.984} C_VEL
LIN {X 0,Y 520.861,Z 597.845,A -85,B 0,C 180,E1 5275.61,E2 5275.61} C_VEL
LIN {X 0,Y 519.481,Z 640.172,A -85,B 0,C 180,E1 5276.639,E2 5276.639} C_VEL
LIN {X 0,Y 517.433,Z 677.434,A -85,B 0,C 180,E1 5278.207,E2 5278.207} C_VEL
LIN {X 0,Y 514.718,Z 714.391,A -85,B 0,C 180,E1 5280.468,E2 5280.468} C_VEL
LIN {X 0,Y 511.949,Z 747.827,A -85,B 0,C 180,E1 5283.287,E2 5283.287} C_VEL
LIN {X 0,Y 509.425,Z 778.247,A -85,B 0,C 180,E1 5286.669,E2 5286.669} C_VEL
LIN {X 0,Y 507.331,Z 805.466,A -85,B 0,C 180,E1 5290.699,E2 5290.699} C_VEL
LIN {X 0,Y 506.08,Z 826.802,A -85,B 0,C 180,E1 5294.969,E2 5294.969} C_VEL
LIN {X 0,Y 505.509,Z 842.084,A -85,B 0,C 180,E1 5299.246,E2 5299.246} C_VEL
LIN {X 0,Y 505.211,Z 851.249,A -85,B 0,C 180,E1 5303.137,E2 5303.137} C_VEL
LIN {X 0,Y 505.166,Z 855.943,A -85,B 0,C 180,E1 5306.574,E2 5306.574} C_VEL
LIN {X 0,Y 505.103,Z 857.5,A -85,B 0,C 180,E1 5309.999,E2 5309.999} C_VEL
LIN {X 0,Y 505.081,Z 855.944,A -85,B 0,C 180,E1 5313.425,E2 5313.425} C_VEL
LIN {X 0,Y 505.226,Z 849.566,A -85,B 0,C 180,E1 5317.723,E2 5317.723} C_VEL
LIN {X 0,Y 505.576,Z 838.011,A -85,B 0,C 180,E1 5322.059,E2 5322.059} C_VEL
LIN {X 0,Y 506.47,Z 820.475,A -85,B 0,C 180,E1 5326.441,E2 5326.441} C_VEL
LIN {X 0,Y 507.878,Z 798.173,A -85,B 0,C 180,E1 5330.508,E2 5330.508} C_VEL
LIN {X 0,Y 510.073,Z 770.342,A -85,B 0,C 180,E1 5334.298,E2 5334.298} C_VEL
LIN {X 0,Y 512.622,Z 739.46,A -85,B 0,C 180,E1 5337.502,E2 5337.502} C_VEL
LIN {X 0,Y 515.615,Z 702.771,A -85,B 0,C 180,E1 5340.333,E2 5340.333} C_VEL
LIN {X 0,Y 518.266,Z 663.399,A -85,B 0,C 180,E1 5342.463,E2 5342.463} C_VEL
LIN {X 0,Y 520.125,Z 626.002,A -85,B 0,C 180,E1 5343.787,E2 5343.787} C_VEL
LIN {X 0,Y 520.255,Z 597.134,A -85,B 0,C 180,E1 5344.448,E2 5344.448} C_VEL
LIN {X 0,Y 504.413,Z 563.28,A -85,B 0,C 180,E1 5346.301,E2 5346.301} C_VEL
LIN {X 0,Y 504.217,Z 563.28,A -85,B 0,C 180,E1 5351.57,E2 5351.57} C_VEL
LIN {X 0,Y 504.229,Z 563.28,A -85,B 0,C 180,E1 5356.506,E2 5356.506} C_VEL
LIN {X 0,Y 504.316,Z 563.28,A -85,B 0,C 180,E1 5361.074,E2 5361.074} C_VEL
LIN {X 0,Y 504.232,Z 563.28,A -85,B 0,C 180,E1 5366.923,E2 5366.923} C_VEL
LIN {X 0,Y 504.41,Z 563.28,A -85,B 0,C 180,E1 5373.339,E2 5373.339} C_VEL
LIN {X 0,Y 504.574,Z 563.28,A -85,B 0,C 180,E1 5378.971,E2 5378.971} C_VEL
LIN {X 0,Y 504.516,Z 563.28,A -85,B 0,C 180,E1 5384.386,E2 5384.386} C_VEL
LIN {X 0,Y 504.672,Z 563.28,A -85,B 0,C 180,E1 5390.649,E2 5390.649} C_VEL
LIN {X 0,Y 504.854,Z 563.28,A -85,B 0,C 180,E1 5396.575,E2 5396.575} C_VEL
LIN {X 0,Y 504.876,Z 563.28,A -85,B 0,C 180,E1 5401.715,E2 5401.715} C_VEL
LIN {X 0,Y 504.78,Z 563.28,A -85,B 0,C 180,E1 5406.869,E2 5406.869} C_VEL
LIN {X 0,Y 504.712,Z 563.28,A -85,B 0,C 180,E1 5412.082,E2 5412.082} C_VEL
LIN {X 0,Y 504.676,Z 563.28,A -85,B 0,C 180,E1 5417.399,E2 5417.399} C_VEL
LIN {X 0,Y 504.514,Z 563.28,A -85,B 0,C 180,E1 5422.883,E2 5422.883} C_VEL
LIN {X 0,Y 504.401,Z 563.28,A -85,B 0,C 180,E1 5428.6,E2 5428.6} C_VEL
LIN {X 0,Y 504.48,Z 563.28,A -85,B 0,C 180,E1 5434.635,E2 5434.635} C_VEL
LIN {X 0,Y 504.27,Z 563.28,A -85,B 0,C 180,E1 5441.175,E2 5441.175} C_VEL
LIN {X 0,Y 504.189,Z 563.28,A -85,B 0,C 180,E1 5446.499,E2 5446.499} C_VEL
LIN {X 0,Y 504.469,Z 563.28,A -85,B 0,C 180,E1 5453.256,E2 5453.256} C_VEL
LIN {X 0,Y 504.488,Z 563.28,A -85,B 0,C 180,E1 5459.437,E2 5459.437} C_VEL
LIN {X 0,Y 504.387,Z 563.28,A -85,B 0,C 180,E1 5465.239,E2 5465.239} C_VEL
LIN {X 0,Y 504.581,Z 563.28,A -85,B 0,C 180,E1 5470.795,E2 5470.795} C_VEL
LIN {X 0,Y 504.791,Z 563.28,A -85,B 0,C 180,E1 5476.164,E2 5476.164} C_VEL
LIN {X 0,Y 504.811,Z 563.28,A -85,B 0,C 180,E1 5481.405,E2 5481.405} C_VEL
LIN {X 0,Y 505.021,Z 563.28,A -85,B 0,C 180,E1 5486.575,E2 5486.575} C_VEL
LIN {X 0,Y 505.119,Z 563.28,A -85,B 0,C 180,E1 5491.713,E2 5491.713} C_VEL
LIN {X 0,Y 504.897,Z 563.28,A -85,B 0,C 180,E1 5496.867,E2 5496.867} C_VEL
LIN {X 0,Y 504.709,Z 563.28,A -85,B 0,C 180,E1 5502.082,E2 5502.082} C_VEL
LIN {X 0,Y 504.643,Z 563.28,A -85,B 0,C 180,E1 5507.4,E2 5507.4} C_VEL
LIN {X 0,Y 504.496,Z 563.28,A -85,B 0,C 180,E1 5512.884,E2 5512.884} C_VEL
LIN {X 0,Y 504.306,Z 563.28,A -85,B 0,C 180,E1 5518.605,E2 5518.605} C_VEL
LIN {X 0,Y 504.331,Z 563.28,A -85,B 0,C 180,E1 5524.647,E2 5524.647} C_VEL
LIN {X 0,Y 504.396,Z 563.28,A -85,B 0,C 180,E1 5528.934,E2 5528.934} C_VEL
LIN {X 0,Y 504.274,Z 563.28,A -85,B 0,C 180,E1 5535.906,E2 5535.906} C_VEL
LIN {X 0,Y 504.347,Z 563.28,A -85,B 0,C 180,E1 5541.072,E2 5541.072} C_VEL
LIN {X 0,Y 504.246,Z 563.28,A -85,B 0,C 180,E1 5546.924,E2 5546.924} C_VEL
LIN {X 0,Y 504.429,Z 563.28,A -85,B 0,C 180,E1 5553.336,E2 5553.336} C_VEL
LIN {X 0,Y 504.598,Z 563.28,A -85,B 0,C 180,E1 5558.968,E2 5558.968} C_VEL
LIN {X 0,Y 504.527,Z 563.28,A -85,B 0,C 180,E1 5564.383,E2 5564.383} C_VEL
LIN {X 0,Y 504.681,Z 563.28,A -85,B 0,C 180,E1 5570.653,E2 5570.653} C_VEL
